C07291=1020.552,377.492,349.340,172.232,49.902,160.000
C07292=1020.561,377.739,349.299,172.241,49.902,160.002
C07293=1020.569,377.985,349.259,172.250,49.901,160.003
C07294=1020.578,378.232,349.218,172.260,49.900,160.005
C07295=1020.587,378.478,349.176,172.269,49.900,160.006
C07296=1020.595,378.724,349.136,172.279,49.900,160.007
C07297=1020.604,378.971,349.094,172.288,49.899,160.009
C07298=1020.613,379.218,349.053,172.297,49.899,160.010
C07299=1020.621,379.464,349.012,172.306,49.899,160.012
C07300=1020.630,379.710,348.971,172.315,49.898,160.013
C07301=1020.639,379.957,348.930,172.325,49.898,160.015
C07302=1020.648,380.203,348.889,172.334,49.898,160.016
C07303=1020.657,380.449,348.847,172.344,49.897,160.018
C07304=1020.665,380.696,348.806,172.353,49.897,160.019
C07305=1020.674,380.943,348.764,172.363,49.897,160.021
C07306=1020.683,381.190,348.723,172.372,49.896,160.022
C07307=1020.693,381.465,348.678,172.383,49.896,160.024
C07308=1020.703,381.741,348.632,172.394,49.896,160.025
C07309=1020.712,382.017,348.585,172.405,49.896,160.027
C07310=1020.723,382.292,348.538,172.415,49.895,160.029
C07311=1020.731,382.539,348.497,172.425,49.895,160.030
C07312=1020.740,382.786,348.455,172.435,49.895,160.032
C07313=1020.750,383.032,348.414,172.444,49.895,160.033
C07314=1020.759,383.278,348.372,172.454,49.894,160.035
C07315=1020.768,383.525,348.331,172.463,49.894,160.036
C07316=1020.777,383.771,348.289,172.473,49.894,160.038
C07317=1020.786,384.017,348.247,172.483,49.894,160.040
C07318=1020.795,384.263,348.206,172.492,49.893,160.041
C07319=1020.804,384.510,348.164,172.503,49.893,160.043
C07320=1020.813,384.756,348.123,172.513,49.893,160.044
C07321=1020.822,385.002,348.081,172.522,49.893,160.046
C07322=1020.831,385.249,348.039,172.532,49.893,160.047
C07323=1020.840,385.495,347.997,172.542,49.893,160.049
C07324=1020.849,385.741,347.955,172.551,49.893,160.051
C07325=1020.859,385.988,347.913,172.562,49.893,160.052
C07326=1020.868,386.234,347.871,172.572,49.893,160.054
C07327=1020.877,386.480,347.829,172.582,49.893,160.056
C07328=1020.886,386.726,347.786,172.592,49.893,160.057
C07329=1020.895,386.972,347.745,172.601,49.893,160.059
C07330=1020.904,387.218,347.702,172.612,49.893,160.060
C07331=1020.914,387.465,347.660,172.622,49.893,160.062
C07332=1020.923,387.711,347.618,172.632,49.893,160.064
C07333=1020.932,387.957,347.576,172.642,49.893,160.066
C07334=1020.941,388.203,347.534,172.652,49.893,160.067
C07335=1020.951,388.449,347.491,172.662,49.894,160.069
C07336=1020.959,388.696,347.449,172.672,49.894,160.071
C07337=1020.969,388.942,347.406,172.682,49.894,160.072
C07338=1020.978,389.188,347.363,172.693,49.894,160.074
C07339=1020.988,389.434,347.321,172.703,49.894,160.076
C07340=1020.996,389.680,347.278,172.713,49.894,160.078
C07341=1021.006,389.926,347.235,172.724,49.894,160.079
C07342=1021.015,390.172,347.193,172.734,49.895,160.081
C07343=1021.025,390.419,347.150,172.744,49.895,160.083
C07344=1021.034,390.664,347.107,172.754,49.895,160.084
C07345=1021.043,390.911,347.064,172.765,49.896,160.086
C07346=1021.053,391.157,347.022,172.776,49.895,160.088
C07347=1021.063,391.403,346.979,172.785,49.896,160.090
C07348=1021.072,391.648,346.936,172.796,49.897,160.092
C07349=1021.081,391.895,346.892,172.807,49.896,160.094
C07350=1021.090,392.141,346.850,172.816,49.897,160.095
C07351=1021.100,392.387,346.807,172.828,49.897,160.097
C07352=1021.110,392.632,346.764,172.838,49.897,160.099
C07353=1021.119,392.879,346.720,172.849,49.898,160.101
C07354=1021.129,393.126,346.678,172.859,49.898,160.103
C07355=1021.138,393.371,346.634,172.870,49.899,160.105
C07356=1021.147,393.618,346.591,172.880,49.899,160.106
C07357=1021.158,393.863,346.548,172.891,49.899,160.108
C07358=1021.166,394.109,346.504,172.902,49.900,160.110
C07359=1021.176,394.355,346.461,172.913,49.901,160.112
C07360=1021.186,394.601,346.417,172.923,49.901,160.114
C07361=1021.195,394.846,346.374,172.934,49.901,160.116
C07362=1021.205,395.093,346.331,172.945,49.902,160.118
C07363=1021.214,395.339,346.287,172.955,49.903,160.120
C07364=1021.225,395.585,346.243,172.967,49.903,160.122
C07365=1021.234,395.831,346.199,172.977,49.904,160.124
C07366=1021.244,396.076,346.156,172.988,49.904,160.125
C07367=1021.256,396.390,346.100,173.002,49.905,160.128
C07368=1021.268,396.703,346.045,173.016,49.906,160.131
C07369=1021.281,397.017,345.989,173.030,49.906,160.133
C07370=1021.294,397.330,345.934,173.044,49.907,160.135
C07371=1021.303,397.576,345.890,173.055,49.907,160.137
C07372=1021.313,397.822,345.845,173.067,49.908,160.140
C07373=1021.323,398.067,345.801,173.078,49.909,160.142
C07374=1021.333,398.313,345.757,173.088,49.910,160.143
C07375=1021.343,398.559,345.714,173.099,49.910,160.145
C07376=1021.352,398.805,345.669,173.111,49.911,160.148
C07377=1021.363,399.051,345.625,173.122,49.912,160.150
C07378=1021.372,399.297,345.581,173.134,49.913,160.152
C07379=1021.382,399.542,345.536,173.144,49.913,160.154
C07380=1021.392,399.788,345.493,173.155,49.914,160.156
C07381=1021.402,400.034,345.448,173.167,49.915,160.158
C07382=1021.412,400.280,345.403,173.179,49.916,160.160
C07383=1021.422,400.526,345.359,173.190,49.916,160.162
C07384=1021.432,400.771,345.314,173.202,49.917,160.164
C07385=1021.441,401.017,345.270,173.213,49.918,160.166
C07386=1021.452,401.263,345.226,173.225,49.919,160.169
C07387=1021.462,401.509,345.181,173.236,49.920,160.171
C07388=1021.472,401.754,345.136,173.248,49.921,160.173
C07389=1021.481,402.000,345.091,173.259,49.922,160.175
C07390=1021.492,402.246,345.046,173.271,49.922,160.177
C07391=1021.501,402.491,345.001,173.282,49.923,160.179
C07392=1021.512,402.737,344.957,173.294,49.924,160.181
C07393=1021.522,402.983,344.912,173.306,49.925,160.184
C07394=1021.532,403.228,344.867,173.317,49.926,160.186
C07395=1021.542,403.475,344.822,173.329,49.927,160.188
C07396=1021.552,403.720,344.777,173.341,49.928,160.190
C07397=1021.563,403.965,344.732,173.352,49.929,160.192
C07398=1021.573,404.211,344.687,173.364,49.931,160.195
C07399=1021.583,404.456,344.642,173.376,49.932,160.197
C07400=1021.593,404.702,344.596,173.388,49.933,160.199
C07401=1021.604,404.948,344.551,173.399,49.934,160.202
C07402=1021.613,405.194,344.506,173.412,49.935,160.204
C07403=1021.625,405.439,344.461,173.424,49.936,160.206
C07404=1021.634,405.684,344.416,173.436,49.937,160.208
C07405=1021.645,405.930,344.370,173.448,49.939,160.211
C07406=1021.655,406.176,344.325,173.460,49.939,160.213
C07407=1021.666,406.422,344.279,173.472,49.941,160.216
C07408=1021.677,406.666,344.234,173.484,49.942,160.218
C07409=1021.687,406.913,344.189,173.496,49.943,160.220
C07410=1021.698,407.158,344.143,173.509,49.944,160.222
C07411=1021.708,407.404,344.097,173.521,49.945,160.225
C07412=1021.719,407.650,344.052,173.533,49.946,160.227
C07413=1021.729,407.895,344.006,173.545,49.948,160.230
C07414=1021.740,408.140,343.961,173.557,49.949,160.232
C07415=1021.751,408.386,343.915,173.570,49.950,160.234
C07416=1021.761,408.631,343.869,173.582,49.951,160.237
C07417=1021.772,408.877,343.823,173.595,49.952,160.239
C07418=1021.782,409.123,343.777,173.607,49.954,160.242
C07419=1021.793,409.368,343.731,173.620,49.955,160.244
C07420=1021.804,409.614,343.686,173.632,49.957,160.246
C07421=1021.815,409.859,343.639,173.645,49.958,160.249
C07422=1021.825,410.104,343.593,173.657,49.959,160.251
C07423=1021.836,410.350,343.547,173.671,49.961,160.254
C07424=1021.846,410.595,343.500,173.683,49.963,160.256
C07425=1021.857,410.841,343.454,173.696,49.964,160.259
C07426=1021.868,411.086,343.407,173.708,49.965,160.261
C07427=1021.881,411.399,343.348,173.724,49.968,160.265
C07428=1021.895,411.712,343.289,173.741,49.969,160.268
C07429=1021.910,412.026,343.230,173.757,49.971,160.271
C07430=1021.923,412.338,343.171,173.773,49.973,160.274
C07431=1021.934,412.584,343.124,173.786,49.975,160.277
C07432=1021.945,412.829,343.077,173.799,49.976,160.280
C07433=1021.956,413.074,343.031,173.813,49.978,160.282
C07434=1021.967,413.320,342.984,173.825,49.979,160.285
C07435=1021.978,413.565,342.937,173.838,49.981,160.287
C07436=1021.989,413.810,342.890,173.852,49.983,160.290
C07437=1022.000,414.055,342.843,173.865,49.984,160.293
C07438=1022.011,414.300,342.797,173.878,49.986,160.295
C07439=1022.022,414.546,342.749,173.892,49.987,160.298
C07440=1022.033,414.791,342.702,173.904,49.989,160.301
C07441=1022.045,415.037,342.655,173.917,49.991,160.303
C07442=1022.056,415.283,342.608,173.931,49.993,160.306
C07443=1022.067,415.528,342.562,173.944,49.994,160.309
C07444=1022.078,415.773,342.514,173.958,49.996,160.312
C07445=1022.089,416.018,342.467,173.971,49.998,160.314
C07446=1022.100,416.263,342.419,173.985,49.999,160.317
C07447=1022.112,416.509,342.372,173.998,50.002,160.320
C07448=1022.122,416.754,342.324,174.012,50.003,160.323
C07449=1022.134,416.999,342.277,174.025,50.005,160.325
C07450=1022.146,417.244,342.229,174.039,50.007,160.328
C07451=1022.156,417.489,342.181,174.052,50.009,160.331
C07452=1022.168,417.735,342.134,174.067,50.011,160.334
C07453=1022.179,417.980,342.086,174.081,50.013,160.337
C07454=1022.191,418.225,342.038,174.094,50.015,160.340
C07455=1022.202,418.470,341.990,174.108,50.016,160.342
C07456=1022.213,418.716,341.942,174.122,50.019,160.345
C07457=1022.225,418.960,341.895,174.136,50.021,160.348
C07458=1022.236,419.205,341.846,174.150,50.022,160.351
C07459=1022.248,419.450,341.799,174.164,50.024,160.354
C07460=1022.259,419.695,341.751,174.177,50.027,160.357
C07461=1022.271,419.941,341.703,174.192,50.028,160.360
C07462=1022.282,420.186,341.655,174.206,50.031,160.363
C07463=1022.294,420.432,341.606,174.221,50.033,160.366
C07464=1022.306,420.676,341.558,174.235,50.035,160.369
C07465=1022.318,420.921,341.510,174.249,50.037,160.372
C07466=1022.329,421.167,341.462,174.263,50.039,160.375
C07467=1022.341,421.411,341.414,174.277,50.041,160.378
C07468=1022.352,421.657,341.365,174.292,50.043,160.381
C07469=1022.365,421.902,341.316,174.306,50.045,160.384
C07470=1022.376,422.147,341.268,174.321,50.047,160.387
C07471=1022.389,422.415,341.215,174.336,50.050,160.390
C07472=1022.402,422.683,341.161,174.352,50.052,160.393
C07473=1022.415,422.951,341.108,174.369,50.054,160.397
C07474=1022.428,423.219,341.055,174.384,50.057,160.400
C07475=1022.439,423.463,341.006,174.399,50.059,160.403
C07476=1022.451,423.709,340.957,174.414,50.062,160.407
C07477=1022.464,423.953,340.908,174.428,50.064,160.410
C07478=1022.476,424.199,340.859,174.443,50.066,160.413
C07479=1022.488,424.443,340.810,174.459,50.068,160.416
C07480=1022.500,424.689,340.761,174.474,50.071,160.419
C07481=1022.511,424.933,340.712,174.488,50.073,160.422
C07482=1022.524,425.178,340.662,174.503,50.076,160.426
C07483=1022.536,425.423,340.613,174.518,50.078,160.429
C07484=1022.548,425.668,340.564,174.534,50.080,160.432
C07485=1022.560,425.913,340.514,174.549,50.083,160.435
C07486=1022.572,426.157,340.466,174.564,50.085,160.439
C07487=1022.588,426.479,340.400,174.584,50.089,160.443
C07488=1022.604,426.800,340.335,174.604,50.091,160.447
C07489=1022.620,427.120,340.269,174.624,50.095,160.452
C07490=1022.636,427.441,340.204,174.644,50.098,160.456
C07491=1022.648,427.685,340.155,174.660,50.101,160.459
C07492=1022.661,427.930,340.105,174.675,50.103,160.463
C07493=1022.673,428.175,340.055,174.691,50.106,160.466
C07494=1022.685,428.420,340.004,174.706,50.109,160.470
C07495=1022.697,428.665,339.954,174.722,50.111,160.473
C07496=1022.710,428.909,339.904,174.738,50.114,160.476
C07497=1022.723,429.154,339.855,174.754,50.116,160.480
C07498=1022.735,429.399,339.805,174.769,50.119,160.483
C07499=1022.747,429.643,339.755,174.785,50.122,160.487
C07500=1022.760,429.888,339.704,174.802,50.125,160.490
C07501=1022.772,430.133,339.654,174.817,50.127,160.494
C07502=1022.785,430.377,339.604,174.834,50.130,160.497
C07503=1022.799,430.622,339.553,174.849,50.133,160.501
C07504=1022.811,430.867,339.503,174.866,50.135,160.504
C07505=1022.824,431.111,339.452,174.881,50.138,160.508
C07506=1022.836,431.355,339.401,174.898,50.141,160.511
C07507=1022.849,431.601,339.351,174.914,50.144,160.515
C07508=1022.862,431.845,339.300,174.931,50.147,160.519
C07509=1022.875,432.089,339.250,174.947,50.149,160.522
C07510=1022.888,432.334,339.199,174.964,50.152,160.526
C07511=1022.901,432.578,339.149,174.980,50.155,160.529
C07512=1022.914,432.823,339.097,174.997,50.158,160.533
C07513=1022.927,433.067,339.046,175.013,50.161,160.537
C07514=1022.939,433.311,338.995,175.030,50.164,160.540
C07515=1022.953,433.556,338.944,175.047,50.166,160.544
C07516=1022.965,433.800,338.893,175.064,50.169,160.548
C07517=1022.978,434.045,338.842,175.081,50.172,160.552
C07518=1022.992,434.289,338.790,175.097,50.176,160.555
C07519=1023.005,434.534,338.739,175.114,50.179,160.559
C07520=1023.018,434.778,338.687,175.131,50.182,160.563
C07521=1023.031,435.023,338.635,175.148,50.185,160.567
C07522=1023.044,435.267,338.584,175.165,50.188,160.571
C07523=1023.057,435.512,338.533,175.182,50.191,160.574
C07524=1023.070,435.756,338.481,175.199,50.194,160.578
C07525=1023.084,436.000,338.429,175.217,50.197,160.582
C07526=1023.097,436.244,338.377,175.235,50.200,160.586
C07527=1023.110,436.488,338.326,175.252,50.203,160.590
C07528=1023.124,436.732,338.274,175.269,50.207,160.594
C07529=1023.137,436.977,338.222,175.286,50.210,160.598
C07530=1023.150,437.221,338.169,175.304,50.212,160.602
C07531=1023.164,437.465,338.117,175.322,50.216,160.606
C07532=1023.177,437.710,338.066,175.339,50.219,160.610
C07533=1023.191,437.954,338.014,175.357,50.222,160.614
C07534=1023.204,438.198,337.961,175.375,50.226,160.618
C07535=1022.814,436.266,338.039,175.226,50.266,160.605
C07536=1022.801,436.022,338.091,175.209,50.264,160.601
C07537=1022.788,435.777,338.142,175.191,50.260,160.597
C07538=1022.774,435.533,338.194,175.174,50.257,160.593
C07539=1022.761,435.289,338.246,175.157,50.254,160.589
C07540=1022.748,435.044,338.297,175.139,50.252,160.585
C07541=1022.735,434.800,338.349,175.122,50.248,160.581
C07542=1022.722,434.556,338.400,175.105,50.245,160.578
C07543=1022.708,434.312,338.451,175.088,50.243,160.574
C07544=1022.695,434.067,338.503,175.071,50.240,160.570
C07545=1022.683,433.823,338.553,175.054,50.237,160.567
C07546=1022.669,433.578,338.605,175.038,50.234,160.563
C07547=1022.656,433.334,338.656,175.021,50.231,160.559
C07548=1022.643,433.089,338.707,175.004,50.228,160.555
C07549=1022.631,432.845,338.758,174.988,50.226,160.552
C07550=1022.618,432.601,338.809,174.971,50.223,160.548
C07551=1022.605,432.356,338.860,174.955,50.220,160.544
C07552=1022.592,432.112,338.911,174.938,50.217,160.541
C07553=1022.579,431.867,338.962,174.922,50.215,160.537
C07554=1022.567,431.622,339.012,174.905,50.212,160.534
C07555=1022.554,431.378,339.063,174.889,50.209,160.530
C07556=1022.540,431.133,339.114,174.873,50.206,160.526
C07557=1022.528,430.888,339.164,174.857,50.204,160.523
C07558=1022.515,430.644,339.214,174.840,50.201,160.519
C07559=1022.503,430.399,339.265,174.825,50.198,160.516
C07560=1022.490,430.154,339.315,174.808,50.196,160.512
C07561=1022.477,429.911,339.365,174.792,50.193,160.509
C07562=1022.464,429.665,339.415,174.776,50.191,160.505
C07563=1022.452,429.420,339.465,174.760,50.188,160.502
C07564=1022.439,429.176,339.516,174.744,50.186,160.499
C07565=1022.427,428.931,339.566,174.729,50.183,160.495
C07566=1022.415,428.686,339.616,174.713,50.180,160.492
C07567=1022.402,428.442,339.666,174.697,50.178,160.488
C07568=1022.390,428.198,339.716,174.681,50.176,160.485
C07569=1022.378,427.953,339.766,174.666,50.173,160.482
C07570=1022.365,427.708,339.816,174.650,50.170,160.478
C07571=1022.353,427.463,339.865,174.635,50.168,160.475
C07572=1022.338,427.163,339.926,174.616,50.165,160.471
C07573=1022.323,426.862,339.988,174.596,50.162,160.467
C07574=1022.308,426.561,340.048,174.578,50.159,160.463
C07575=1022.294,426.261,340.110,174.559,50.156,160.458
C07576=1022.281,426.016,340.159,174.543,50.154,160.455
C07577=1022.269,425.771,340.208,174.528,50.152,160.452
C07578=1022.257,425.526,340.258,174.513,50.149,160.449
C07579=1022.245,425.281,340.308,174.498,50.147,160.445
C07580=1022.233,425.037,340.356,174.483,50.145,160.442
C07581=1022.221,424.791,340.406,174.468,50.143,160.439
C07582=1022.209,424.546,340.455,174.454,50.140,160.436
C07583=1022.197,424.301,340.503,174.438,50.138,160.433
C07584=1022.185,424.057,340.552,174.424,50.136,160.430
C07585=1022.172,423.811,340.601,174.408,50.134,160.426
C07586=1022.161,423.567,340.650,174.394,50.132,160.423
C07587=1022.149,423.321,340.700,174.379,50.129,160.420
C07588=1022.137,423.077,340.748,174.364,50.127,160.417
C07589=1022.125,422.832,340.797,174.349,50.125,160.414
C07590=1022.113,422.587,340.846,174.335,50.123,160.411
C07591=1022.102,422.342,340.894,174.321,50.121,160.408
C07592=1022.090,422.097,340.943,174.305,50.119,160.405
C07593=1022.078,421.852,340.992,174.292,50.116,160.402
C07594=1022.067,421.607,341.040,174.277,50.115,160.399
C07595=1022.055,421.362,341.089,174.263,50.112,160.396
C07596=1022.043,421.116,341.137,174.248,50.111,160.393
C07597=1022.031,420.872,341.185,174.234,50.108,160.390
C07598=1022.020,420.627,341.234,174.220,50.107,160.387
C07599=1022.008,420.382,341.281,174.206,50.104,160.384
C07600=1021.996,420.137,341.329,174.191,50.103,160.381
C07601=1021.985,419.891,341.377,174.177,50.100,160.378
C07602=1021.973,419.647,341.426,174.163,50.099,160.375
C07603=1021.962,419.401,341.474,174.149,50.097,160.372
C07604=1021.950,419.156,341.522,174.135,50.095,160.369
C07605=1021.938,418.911,341.570,174.121,50.093,160.366
C07606=1021.927,418.666,341.618,174.107,50.091,160.364
C07607=1021.916,418.420,341.665,174.093,50.090,160.361
C07608=1021.904,418.175,341.713,174.078,50.088,160.358
C07609=1021.893,417.930,341.761,174.065,50.086,160.355
C07610=1021.881,417.685,341.808,174.051,50.084,160.352
C07611=1021.870,417.440,341.856,174.038,50.082,160.349
C07612=1021.859,417.194,341.903,174.024,50.081,160.347
C07613=1021.848,416.949,341.952,174.010,50.079,160.344
C07614=1021.837,416.704,341.998,173.996,50.077,160.341
C07615=1021.825,416.459,342.046,173.983,50.075,160.338
C07616=1021.814,416.213,342.094,173.969,50.074,160.335
C07617=1021.803,415.969,342.141,173.956,50.072,160.333
C07618=1021.792,415.723,342.189,173.942,50.070,160.330
C07619=1021.780,415.478,342.236,173.929,50.069,160.327
C07620=1021.764,415.118,342.305,173.909,50.066,160.323
C07621=1021.748,414.757,342.375,173.890,50.064,160.319
C07622=1021.731,414.397,342.443,173.870,50.062,160.315
C07623=1021.715,414.036,342.512,173.851,50.059,160.311
C07624=1021.704,413.791,342.559,173.838,50.057,160.309
C07625=1021.693,413.546,342.606,173.825,50.056,160.306
C07626=1021.682,413.301,342.652,173.811,50.054,160.304
C07627=1021.671,413.056,342.699,173.798,50.053,160.301
C07628=1021.660,412.821,342.744,173.786,50.051,160.298
C07629=1021.650,412.587,342.788,173.773,50.050,160.296
C07630=1021.639,412.352,342.833,173.761,50.049,160.293
C07631=1021.629,412.118,342.878,173.749,50.047,160.291
C07632=1021.619,411.884,342.922,173.736,50.046,160.289
C07633=1021.608,411.648,342.966,173.724,50.045,160.286
C07634=1021.598,411.414,343.010,173.712,50.044,160.284
C07635=1021.588,411.180,343.055,173.700,50.042,160.281
C07636=1021.578,410.935,343.101,173.687,50.041,160.279
C07637=1021.567,410.690,343.147,173.673,50.039,160.276
C07638=1021.555,410.443,343.194,173.661,50.038,160.274
C07639=1021.545,410.198,343.240,173.648,50.037,160.271
C07640=1021.534,409.953,343.286,173.636,50.035,160.269
C07641=1021.524,409.707,343.333,173.623,50.034,160.266
C07642=1021.513,409.461,343.379,173.610,50.033,160.264
C07643=1021.502,409.216,343.425,173.598,50.031,160.261
C07644=1021.492,408.971,343.471,173.585,50.030,160.259
C07645=1021.481,408.725,343.517,173.573,50.029,160.257
C07646=1021.471,408.479,343.562,173.560,50.028,160.254
C07647=1021.460,408.234,343.608,173.548,50.026,160.252
C07648=1021.449,407.988,343.653,173.536,50.026,160.250
C07649=1021.438,407.742,343.699,173.524,50.024,160.247
C07650=1021.428,407.497,343.745,173.511,50.023,160.245
C07651=1021.418,407.252,343.791,173.499,50.022,160.242
C07652=1021.407,407.006,343.836,173.487,50.021,160.240
C07653=1021.396,406.760,343.881,173.474,50.020,160.238
C07654=1021.385,406.515,343.927,173.463,50.019,160.235
C07655=1021.376,406.269,343.972,173.451,50.018,160.233
C07656=1021.365,406.024,344.018,173.438,50.017,160.231
C07657=1021.355,405.777,344.063,173.426,50.016,160.229
C07658=1021.344,405.533,344.108,173.414,50.014,160.226
C07659=1021.334,405.287,344.153,173.402,50.014,160.224
C07660=1021.323,405.041,344.199,173.390,50.013,160.222
C07661=1021.313,404.796,344.244,173.378,50.012,160.219
C07662=1021.303,404.549,344.289,173.367,50.011,160.217
C07663=1021.292,404.305,344.334,173.353,50.010,160.215
C07664=1021.282,404.059,344.379,173.342,50.009,160.212
C07665=1021.272,403.813,344.424,173.330,50.008,160.210
C07666=1021.262,403.567,344.469,173.318,50.007,160.208
C07667=1021.252,403.321,344.514,173.307,50.006,160.206
C07668=1021.242,403.076,344.558,173.295,50.005,160.204
C07669=1021.231,402.830,344.604,173.284,50.004,160.202
C07670=1021.221,402.585,344.649,173.271,50.004,160.199
C07671=1021.212,402.339,344.694,173.260,50.003,160.197
C07672=1021.201,402.093,344.739,173.248,50.002,160.195
C07673=1021.192,401.847,344.783,173.236,50.001,160.193
C07674=1021.181,401.602,344.827,173.225,50.000,160.191
C07675=1021.171,401.356,344.873,173.213,49.999,160.189
C07676=1021.161,401.110,344.917,173.202,49.998,160.186
C07677=1021.152,400.865,344.962,173.190,49.998,160.184
C07678=1021.142,400.619,345.006,173.179,49.997,160.182
C07679=1021.132,400.373,345.051,173.167,49.996,160.180
C07680=1021.122,400.127,345.096,173.156,49.995,160.178
C07681=1021.111,399.881,345.139,173.145,49.995,160.176
C07682=1021.102,399.636,345.184,173.134,49.994,160.174
C07683=1021.092,399.390,345.228,173.123,49.993,160.172
C07684=1021.082,399.144,345.273,173.111,49.993,160.170
C07685=1021.072,398.898,345.317,173.100,49.992,160.168
C07686=1021.062,398.652,345.360,173.088,49.991,160.166
C07687=1021.053,398.407,345.405,173.077,49.991,160.164
C07688=1021.043,398.161,345.449,173.066,49.991,160.162
C07689=1021.033,397.915,345.493,173.055,49.990,160.160
C07690=1021.024,397.669,345.537,173.044,49.989,160.158
C07691=1021.013,397.423,345.580,173.033,49.988,160.155
C07692=1021.001,397.108,345.637,173.019,49.988,160.153
C07693=1020.988,396.792,345.694,173.004,49.987,160.150
C07694=1020.975,396.477,345.749,172.990,49.986,160.148
C07695=1020.963,396.161,345.805,172.976,49.986,160.146
C07696=1020.953,395.915,345.848,172.965,49.986,160.144
C07697=1020.944,395.669,345.892,172.954,49.985,160.142
C07698=1020.934,395.424,345.936,172.943,49.984,160.140
C07699=1020.925,395.177,345.980,172.932,49.985,160.138
C07700=1020.914,394.932,346.023,172.921,49.984,160.136
C07701=1020.905,394.685,346.066,172.911,49.983,160.134
C07702=1020.896,394.440,346.110,172.900,49.983,160.132
C07703=1020.886,394.194,346.153,172.889,49.983,160.130
C07704=1020.877,393.947,346.197,172.878,49.982,160.128
C07705=1020.867,393.702,346.240,172.868,49.982,160.126
C07706=1020.857,393.456,346.283,172.857,49.981,160.125
C07707=1020.848,393.209,346.327,172.846,49.982,160.123
C07708=1020.839,392.964,346.369,172.836,49.981,160.121
C07709=1020.829,392.718,346.413,172.825,49.981,160.119
C07710=1020.820,392.472,346.456,172.814,49.981,160.117
C07711=1020.810,392.225,346.498,172.804,49.980,160.115
C07712=1020.800,391.979,346.541,172.793,49.980,160.114
C07713=1020.791,391.734,346.585,172.783,49.980,160.112
C07714=1020.782,391.487,346.628,172.772,49.980,160.110
C07715=1020.772,391.241,346.670,172.762,49.979,160.108
C07716=1020.762,390.995,346.713,172.751,49.980,160.106
C07717=1020.754,390.749,346.756,172.741,49.979,160.105
C07718=1020.744,390.502,346.799,172.731,49.979,160.103
C07719=1020.735,390.257,346.841,172.720,49.979,160.101
C07720=1020.726,390.011,346.884,172.711,49.979,160.100
C07721=1020.716,389.764,346.926,172.699,49.978,160.098
C07722=1020.707,389.518,346.970,172.689,49.978,160.096
C07723=1020.697,389.272,347.012,172.679,49.978,160.094
C07724=1020.688,389.026,347.055,172.669,49.979,160.093
C07725=1020.679,388.780,347.097,172.659,49.978,160.091
C07726=1020.671,388.534,347.139,172.648,49.979,160.089
C07727=1020.661,388.287,347.182,172.638,49.978,160.087
C07728=1020.652,388.042,347.225,172.628,49.978,160.086
C07729=1020.643,387.795,347.266,172.617,49.978,160.084
C07730=1020.633,387.549,347.309,172.608,49.979,160.082
C07731=1020.624,387.303,347.352,172.598,49.978,160.081
C07732=1020.615,387.057,347.393,172.588,49.978,160.079
C07733=1020.606,386.811,347.436,172.578,49.979,160.077
C07734=1020.597,386.565,347.478,172.568,49.979,160.076
C07735=1020.588,386.318,347.519,172.558,49.978,160.074
C07736=1020.578,386.072,347.562,172.547,49.979,160.073
C07737=1020.569,385.825,347.604,172.537,49.979,160.071
C07738=1020.560,385.580,347.646,172.528,49.979,160.069
C07739=1020.551,385.333,347.688,172.518,49.979,160.068
C07740=1020.542,385.087,347.730,172.508,49.979,160.066
C07741=1020.533,384.841,347.771,172.498,49.980,160.065
C07742=1020.524,384.594,347.813,172.488,49.980,160.063
C07743=1020.515,384.348,347.855,172.479,49.980,160.061
C07744=1020.505,384.102,347.896,172.469,49.980,160.060
C07745=1020.496,383.855,347.938,172.459,49.980,160.058
C07746=1020.487,383.609,347.979,172.449,49.981,160.057
C07747=1020.478,383.363,348.021,172.439,49.981,160.055
C07748=1020.470,383.116,348.063,172.430,49.981,160.054
C07749=1020.461,382.870,348.104,172.420,49.982,160.052
C07750=1020.451,382.624,348.146,172.411,49.982,160.051
C07751=1020.442,382.378,348.187,172.401,49.982,160.049
C07752=1020.432,382.100,348.234,172.390,49.983,160.047
C07753=1020.423,381.821,348.280,172.379,49.983,160.046
C07754=1020.412,381.542,348.327,172.368,49.984,160.044
C07755=1020.402,381.264,348.374,172.357,49.984,160.042
C07756=1020.393,381.018,348.416,172.347,49.984,160.041
C07757=1020.385,380.771,348.456,172.338,49.984,160.039
C07758=1020.375,380.525,348.497,172.329,49.985,160.038
C07759=1020.366,380.279,348.539,172.319,49.986,160.036
C07760=1020.358,380.032,348.580,172.310,49.986,160.035
C07761=1020.349,379.786,348.621,172.300,49.986,160.033
C07762=1020.341,379.539,348.662,172.291,49.987,160.032
C07763=1020.331,379.293,348.703,172.281,49.988,160.031
C07764=1020.323,379.047,348.744,172.272,49.988,160.029
C07765=1020.315,378.800,348.785,172.262,49.988,160.028
C07766=1020.306,378.554,348.827,172.253,49.989,160.026
C07767=1020.298,378.307,348.868,172.245,49.989,160.025
C07768=1020.289,378.060,348.909,172.235,49.989,160.023
C07769=1020.280,377.814,348.949,172.226,49.990,160.022
C07770=1020.271,377.568,348.990,172.216,49.991,160.021
C07771=1020.263,377.322,349.031,172.207,49.991,160.019
C07772=1020.255,377.075,349.072,172.198,49.992,160.018
C07773=1020.247,376.828,349.113,172.188,49.992,160.016
C07774=1020.237,376.582,349.153,172.179,49.993,160.015
C07775=1020.229,376.335,349.194,172.171,49.994,160.014
C07776=1020.220,376.089,349.235,172.161,49.994,160.012
C07777=1020.212,375.842,349.275,172.152,49.995,160.011
C07778=1020.203,375.595,349.316,172.143,49.995,160.010
C07779=1020.194,375.350,349.356,172.134,49.996,160.008
C07780=1020.186,375.103,349.397,172.125,49.997,160.007
C07781=1020.177,374.857,349.437,172.115,49.998,160.006
C07782=1020.169,374.609,349.477,172.107,49.999,160.005
C07783=1020.160,374.363,349.517,172.098,49.999,160.003
C07784=1020.152,374.117,349.558,172.089,50.000,160.002
C07785=1020.143,373.869,349.597,172.079,50.001,160.001
C07786=1020.135,373.623,349.638,172.070,50.002,159.999
C07787=1020.126,373.377,349.678,172.062,50.002,159.998
C07788=1020.118,373.130,349.718,172.053,50.003,159.997
C07789=1020.109,372.884,349.758,172.044,50.004,159.996
C07790=1020.101,372.637,349.798,172.035,50.005,159.994
C07791=1020.092,372.390,349.839,172.027,50.006,159.993
C07792=1020.083,372.143,349.878,172.017,50.007,159.992
C07793=1020.075,371.897,349.919,172.008,50.007,159.990
C07794=1020.067,371.651,349.958,172.000,50.008,159.989
C07795=1020.059,371.404,349.998,171.991,50.009,159.988
C07796=1020.050,371.157,350.038,171.982,50.010,159.987
C07797=1020.042,370.910,350.078,171.973,50.011,159.986
C07798=1020.034,370.663,350.118,171.965,50.012,159.984
C07799=1020.026,370.417,350.158,171.956,50.013,159.983
C07800=1020.017,370.171,350.198,171.947,50.014,159.982
C07801=1020.009,369.924,350.237,171.939,50.015,159.981
C07802=1020.001,369.677,350.277,171.930,50.016,159.980
C07803=1019.993,369.430,350.317,171.922,50.016,159.978
C07804=1019.985,369.184,350.356,171.913,50.018,159.977
C07805=1019.976,368.938,350.396,171.904,50.019,159.976
C07806=1019.968,368.691,350.436,171.896,50.019,159.975
C07807=1019.960,368.444,350.475,171.887,50.021,159.974
C07808=1019.952,368.197,350.515,171.879,50.021,159.973
C07809=1019.944,367.951,350.555,171.870,50.023,159.971
C07810=1019.936,367.704,350.594,171.861,50.024,159.970
C07811=1019.928,367.456,350.633,171.853,50.025,159.969
C07812=1019.918,367.200,350.674,171.844,50.026,159.968
C07813=1019.910,366.945,350.715,171.835,50.028,159.967
C07814=1019.902,366.689,350.756,171.826,50.029,159.966
C07815=1019.894,366.433,350.796,171.817,50.030,159.964
C07816=1019.885,366.186,350.835,171.809,50.031,159.963
C07817=1019.877,365.939,350.874,171.801,50.033,159.962
C07818=1019.869,365.692,350.913,171.792,50.033,159.961
C07819=1019.860,365.445,350.952,171.784,50.035,159.960
C07820=1019.852,365.199,350.992,171.776,50.036,159.959
C07821=1019.844,364.951,351.030,171.767,50.037,159.958
C07822=1019.835,364.705,351.069,171.759,50.039,159.957
C07823=1019.828,364.458,351.108,171.750,50.039,159.956
C07824=1019.820,364.211,351.148,171.742,50.041,159.955
C07825=1019.812,363.964,351.186,171.734,50.042,159.954
C07826=1019.804,363.717,351.225,171.726,50.043,159.953
C07827=1019.796,363.471,351.264,171.717,50.045,159.952
C07828=1019.788,363.224,351.302,171.709,50.046,159.951
C07829=1019.780,362.977,351.341,171.701,50.048,159.950
C07830=1019.772,362.731,351.380,171.693,50.049,159.949
C07831=1019.764,362.483,351.419,171.684,50.050,159.947
C07832=1019.756,362.236,351.458,171.676,50.051,159.946
C07833=1019.749,361.989,351.496,171.667,50.053,159.945
C07834=1019.740,361.743,351.535,171.660,50.054,159.944
C07835=1019.732,361.496,351.574,171.652,50.056,159.944
C07836=1019.724,361.249,351.612,171.644,50.057,159.943
C07837=1019.716,361.002,351.651,171.636,50.059,159.942
C07838=1019.709,360.755,351.689,171.627,50.060,159.940
C07839=1019.701,360.508,351.728,171.619,50.061,159.939
C07840=1019.693,360.261,351.767,171.611,50.062,159.938
C07841=1019.686,360.014,351.805,171.603,50.064,159.938
C07842=1019.677,359.767,351.844,171.595,50.066,159.937
C07843=1019.670,359.520,351.882,171.588,50.067,159.936
C07844=1019.662,359.273,351.921,171.579,50.069,159.935
C07845=1019.654,359.027,351.959,171.571,50.070,159.934
C07846=1019.646,358.779,351.997,171.564,50.072,159.933
C07847=1019.638,358.533,352.034,171.555,50.073,159.932
C07848=1019.631,358.286,352.073,171.547,50.075,159.931
C07849=1019.622,358.039,352.111,171.539,50.077,159.930
C07850=1019.615,357.792,352.149,171.531,50.078,159.929
C07851=1019.607,357.545,352.187,171.524,50.080,159.928
C07852=1019.599,357.298,352.226,171.515,50.082,159.927
C07853=1019.591,357.050,352.263,171.508,50.083,159.926
C07854=1019.583,356.804,352.301,171.500,50.085,159.926
C07855=1019.576,356.557,352.339,171.492,50.086,159.924
C07856=1019.568,356.310,352.377,171.484,50.088,159.924
C07857=1019.560,356.063,352.415,171.477,50.090,159.923
C07858=1019.552,355.816,352.452,171.469,50.091,159.922
C07859=1019.545,355.568,352.490,171.461,50.093,159.921
C07860=1019.537,355.322,352.529,171.453,50.095,159.920
C07861=1019.530,355.075,352.566,171.446,50.097,159.919
C07862=1019.522,354.828,352.605,171.437,50.098,159.918
C07863=1019.514,354.581,352.642,171.430,50.100,159.917
C07864=1019.506,354.334,352.679,171.422,50.102,159.917
C07865=1019.499,354.087,352.717,171.415,50.104,159.916
C07866=1019.492,353.840,352.755,171.406,50.106,159.915
C07867=1019.483,353.592,352.792,171.399,50.107,159.914
C07868=1019.476,353.345,352.830,171.392,50.109,159.913
C07869=1019.468,353.098,352.867,171.384,50.111,159.913
C07870=1019.460,352.851,352.904,171.376,50.113,159.912
C07871=1019.453,352.605,352.942,171.368,50.115,159.911
C07872=1019.445,352.356,352.980,171.361,50.117,159.910
C07873=1019.437,352.107,353.017,171.354,50.118,159.909
C07874=1019.429,351.858,353.055,171.345,50.121,159.909
C07875=1019.422,351.609,353.092,171.338,50.122,159.908
C07876=1019.414,351.362,353.129,171.330,50.124,159.907
C07877=1019.407,351.115,353.167,171.323,50.126,159.906
C07878=1019.399,350.868,353.204,171.315,50.128,159.905
C07879=1019.392,350.621,353.241,171.307,50.130,159.904
C07880=1019.384,350.374,353.278,171.300,50.132,159.904
C07881=1019.377,350.127,353.316,171.293,50.134,159.903
C07882=1019.369,349.880,353.353,171.286,50.136,159.902
C07883=1019.362,349.633,353.390,171.278,50.138,159.901
C07884=1019.354,349.386,353.427,171.270,50.140,159.901
C07885=1019.347,349.139,353.464,171.263,50.142,159.900
C07886=1019.339,348.892,353.502,171.255,50.144,159.899
C07887=1019.332,348.644,353.538,171.248,50.146,159.898
C07888=1019.324,348.397,353.575,171.241,50.148,159.898
C07889=1019.317,348.150,353.613,171.233,50.150,159.897
C07890=1019.309,347.902,353.649,171.226,50.152,159.896
C07891=1019.302,347.655,353.687,171.218,50.154,159.896
C07892=1019.295,347.408,353.723,171.211,50.156,159.895
C07893=1019.287,347.161,353.760,171.204,50.159,159.894
C07894=1019.280,346.915,353.797,171.196,50.160,159.893
C07895=1019.273,346.667,353.834,171.189,50.163,159.893
C07896=1019.265,346.419,353.870,171.182,50.165,159.892
C07897=1019.257,346.173,353.907,171.175,50.167,159.891
C07898=1019.250,345.925,353.944,171.168,50.169,159.891
C07899=1019.243,345.677,353.980,171.159,50.171,159.890
C07900=1019.235,345.431,354.016,171.152,50.174,159.889
C07901=1019.228,345.184,354.053,171.145,50.176,159.889
C07902=1019.221,344.936,354.089,171.138,50.178,159.888
C07903=1019.213,344.689,354.126,171.131,50.181,159.887
C07904=1019.206,344.442,354.163,171.124,50.183,159.887
C07905=1019.199,344.195,354.199,171.117,50.185,159.886
C07906=1019.191,343.947,354.235,171.110,50.187,159.885
C07907=1019.184,343.700,354.272,171.103,50.190,159.885
C07908=1019.177,343.453,354.308,171.096,50.192,159.884
C07909=1019.169,343.206,354.345,171.088,50.194,159.883
C07910=1019.161,342.959,354.381,171.081,50.196,159.883
C07911=1019.155,342.712,354.418,171.073,50.199,159.882
C07912=1019.147,342.464,354.454,171.066,50.201,159.882
C07913=1019.140,342.217,354.490,171.059,50.204,159.881
C07914=1019.133,341.970,354.526,171.052,50.206,159.880
C07915=1019.126,341.722,354.563,171.045,50.209,159.880
C07916=1019.118,341.475,354.599,171.038,50.211,159.879
C07917=1019.111,341.227,354.634,171.031,50.213,159.879
C07918=1019.104,340.980,354.670,171.024,50.216,159.878
C07919=1019.097,340.733,354.707,171.017,50.218,159.877
C07920=1019.090,340.485,354.743,171.010,50.221,159.877
C07921=1019.082,340.239,354.779,171.003,50.223,159.876
C07922=1019.075,339.991,354.815,170.996,50.225,159.876
C07923=1019.069,339.743,354.851,170.989,50.228,159.875
C07924=1019.061,339.496,354.887,170.982,50.230,159.874
C07925=1019.054,339.249,354.923,170.975,50.233,159.874
C07926=1019.046,339.002,354.959,170.968,50.235,159.873
C07927=1019.040,338.754,354.994,170.961,50.237,159.873
C07928=1019.032,338.507,355.030,170.954,50.240,159.872
C07929=1019.025,338.260,355.065,170.947,50.243,159.872
C07930=1019.017,338.012,355.102,170.940,50.245,159.871
C07931=1019.011,337.765,355.137,170.933,50.248,159.870
C07932=1019.003,337.513,355.174,170.926,50.251,159.870
C07933=1018.995,337.262,355.210,170.919,50.253,159.869
C07934=1018.989,337.010,355.246,170.912,50.256,159.869
C07935=1018.981,336.759,355.282,170.905,50.259,159.868
C07936=1018.974,336.512,355.317,170.899,50.261,159.868
C07937=1018.967,336.265,355.353,170.892,50.264,159.867
C07938=1018.960,336.017,355.389,170.885,50.267,159.867
C07939=1018.953,335.770,355.424,170.878,50.269,159.866
C07940=1018.946,335.523,355.460,170.871,50.272,159.866
C07941=1018.938,335.275,355.495,170.864,50.274,159.865
C07942=1018.932,335.027,355.530,170.858,50.277,159.865
C07943=1018.925,334.780,355.565,170.851,50.280,159.864
C07944=1018.917,334.533,355.602,170.844,50.283,159.864
C07945=1018.910,334.285,355.637,170.837,50.285,159.863
C07946=1018.904,334.038,355.672,170.830,50.288,159.863
C07947=1018.897,333.790,355.707,170.823,50.291,159.862
C07948=1018.890,333.542,355.742,170.817,50.294,159.862
C07949=1018.882,333.296,355.778,170.810,50.297,159.861
C07950=1018.876,333.048,355.813,170.803,50.299,159.861
C07951=1018.869,332.801,355.849,170.797,50.302,159.860
C07952=1018.861,332.554,355.883,170.789,50.305,159.860
C07953=1018.854,332.306,355.919,170.783,50.308,159.859
C07954=1018.847,332.058,355.954,170.776,50.311,159.859
C07955=1018.841,331.811,355.989,170.770,50.314,159.859
C07956=1018.833,331.564,356.023,170.763,50.317,159.858
C07957=1018.826,331.317,356.059,170.757,50.319,159.858
C07958=1018.820,331.069,356.093,170.750,50.322,159.857
C07959=1018.812,330.821,356.128,170.744,50.325,159.857
C07960=1018.805,330.574,356.163,170.737,50.328,159.857
C07961=1018.798,330.326,356.198,170.730,50.331,159.856
C07962=1018.791,330.079,356.233,170.724,50.334,159.856
C07963=1018.784,329.831,356.267,170.717,50.337,159.855
C07964=1018.777,329.584,356.302,170.710,50.340,159.855
C07965=1018.771,329.336,356.337,170.703,50.343,159.854
C07966=1018.763,329.089,356.372,170.697,50.346,159.854
C07967=1018.757,328.841,356.406,170.690,50.349,159.854
C07968=1018.750,328.594,356.442,170.684,50.352,159.853
C07969=1018.743,328.347,356.477,170.678,50.355,159.853
C07970=1018.736,328.099,356.510,170.671,50.358,159.852
C07971=1018.729,327.852,356.546,170.665,50.361,159.852
C07972=1018.723,327.604,356.580,170.658,50.364,159.852
C07973=1018.715,327.357,356.615,170.651,50.367,159.851
C07974=1018.708,327.109,356.650,170.645,50.371,159.851
C07975=1018.702,326.861,356.684,170.638,50.374,159.851
C07976=1018.694,326.614,356.719,170.632,50.377,159.850
C07977=1018.688,326.366,356.753,170.626,50.379,159.850
C07978=1018.681,326.119,356.787,170.620,50.383,159.850
C07979=1018.675,325.872,356.822,170.613,50.386,159.849
C07980=1018.667,325.624,356.855,170.607,50.389,159.849
C07981=1018.660,325.377,356.889,170.600,50.392,159.849
C07982=1018.653,325.129,356.923,170.593,50.395,159.848
C07983=1018.646,324.881,356.958,170.587,50.399,159.848
C07984=1018.639,324.634,356.992,170.581,50.402,159.848
C07985=1018.632,324.386,357.026,170.574,50.406,159.847
C07986=1018.625,324.138,357.060,170.568,50.409,159.847
C07987=1018.618,323.890,357.094,170.561,50.412,159.847
C07988=1018.612,323.643,357.128,170.555,50.416,159.846
C07989=1018.604,323.396,357.161,170.548,50.419,159.846
C07990=1018.598,323.148,357.197,170.543,50.422,159.846
C07991=1018.590,322.901,357.230,170.536,50.425,159.846
C07992=1018.583,322.645,357.265,170.529,50.429,159.845
C07993=1018.576,322.389,357.300,170.522,50.432,159.845
C07994=1018.569,322.134,357.335,170.516,50.436,159.845
C07995=1018.562,321.878,357.370,170.510,50.440,159.844
C07996=1018.555,321.631,357.404,170.503,50.443,159.844
C07997=1018.548,321.383,357.438,170.497,50.447,159.844
C07998=1018.542,321.136,357.472,170.490,50.450,159.843
C07999=1018.535,320.887,357.505,170.485,50.453,159.843
C08000=1018.528,320.640,357.539,170.479,50.457,159.843
C08001=1018.521,320.392,357.573,170.472,50.460,159.843
C08002=1018.515,320.145,357.607,170.466,50.463,159.843
C08003=1018.507,319.897,357.640,170.460,50.467,159.842
C08004=1018.501,319.650,357.674,170.453,50.470,159.842
C08005=1018.494,319.402,357.707,170.447,50.474,159.842
C08006=1018.488,319.154,357.741,170.442,50.477,159.842
C08007=1018.481,318.907,357.775,170.435,50.480,159.841
C08008=1018.474,318.659,357.809,170.429,50.484,159.841
C08009=1018.467,318.411,357.843,170.422,50.488,159.841
C08010=1018.461,318.164,357.876,170.416,50.492,159.841
C08011=1018.454,317.916,357.910,170.409,50.495,159.840
C08012=1018.447,317.669,357.943,170.404,50.498,159.840
C08013=1018.440,317.421,357.976,170.398,50.502,159.840
C08014=1018.434,317.173,358.010,170.392,50.505,159.840
C08015=1018.427,316.926,358.044,170.386,50.509,159.840
C08016=1018.421,316.678,358.077,170.379,50.513,159.839
C08017=1018.414,316.430,358.111,170.373,50.517,159.839
C08018=1018.408,316.182,358.144,170.367,50.519,159.839
C08019=1018.401,315.935,358.178,170.361,50.523,159.839
C08020=1018.395,315.687,358.211,170.355,50.527,159.838
C08021=1018.387,315.439,358.244,170.349,50.530,159.838
C08022=1018.381,315.192,358.277,170.342,50.534,159.838
C08023=1018.375,314.945,358.311,170.337,50.537,159.838
C08024=1018.368,314.696,358.344,170.331,50.541,159.838
C08025=1018.362,314.449,358.378,170.325,50.545,159.837
C08026=1018.355,314.201,358.411,170.318,50.549,159.837
C08027=1018.349,313.954,358.445,170.312,50.552,159.837
C08028=1018.343,313.706,358.478,170.307,50.556,159.837
C08029=1018.336,313.459,358.512,170.301,50.559,159.837
C08030=1018.329,313.211,358.544,170.294,50.563,159.837
C08031=1018.323,312.963,358.577,170.289,50.568,159.837
C08032=1018.317,312.715,358.611,170.282,50.571,159.836
C08033=1018.310,312.468,358.644,170.277,50.575,159.836
C08034=1018.304,312.220,358.677,170.271,50.578,159.836
C08035=1018.297,311.973,358.710,170.265,50.582,159.836
C08036=1018.290,311.725,358.743,170.258,50.586,159.836
C08037=1018.285,311.477,358.777,170.253,50.589,159.835
C08038=1018.279,311.229,358.810,170.247,50.594,159.835
C08039=1018.272,310.982,358.843,170.241,50.597,159.835
C08040=1018.265,310.734,358.876,170.235,50.601,159.835
C08041=1018.260,310.486,358.909,170.229,50.604,159.835
C08042=1018.253,310.239,358.942,170.223,50.608,159.835
C08043=1018.247,309.991,358.975,170.217,50.613,159.835
C08044=1018.241,309.743,359.008,170.211,50.616,159.835
C08045=1018.234,309.496,359.040,170.206,50.620,159.834
C08046=1018.227,309.248,359.073,170.200,50.624,159.834
C08047=1018.220,309.000,359.106,170.194,50.628,159.834
C08048=1018.213,308.753,359.138,170.188,50.632,159.834
C08049=1018.207,308.505,359.171,170.182,50.637,159.834
C08050=1018.201,308.257,359.203,170.176,50.640,159.834
C08051=1018.194,308.009,359.235,170.170,50.645,159.834
C08052=1018.187,307.759,359.268,170.164,50.648,159.834
C08053=1018.180,307.509,359.301,170.158,50.653,159.834
C08054=1018.174,307.258,359.333,170.153,50.657,159.834
C08055=1018.167,307.009,359.366,170.147,50.661,159.834
C08056=1018.161,306.761,359.398,170.141,50.665,159.834
C08057=1018.153,306.513,359.430,170.135,50.669,159.834
C08058=1018.147,306.265,359.463,170.129,50.673,159.833
C08059=1018.141,306.017,359.495,170.123,50.677,159.833
C08060=1018.134,305.769,359.527,170.117,50.682,159.833
C08061=1018.128,305.521,359.559,170.112,50.686,159.834
C08062=1018.121,305.274,359.592,170.106,50.690,159.833
C08063=1018.115,305.026,359.624,170.100,50.694,159.833
C08064=1018.108,304.778,359.656,170.094,50.698,159.833
C08065=1018.102,304.531,359.688,170.088,50.703,159.833
C08066=1018.096,304.283,359.721,170.082,50.707,159.833
C08067=1018.089,304.035,359.753,170.077,50.711,159.833
C08068=1018.083,303.787,359.785,170.071,50.715,159.833
C08069=1018.076,303.539,359.816,170.066,50.719,159.833
C08070=1018.070,303.292,359.849,170.060,50.724,159.833
C08071=1018.063,303.044,359.880,170.054,50.728,159.833
C08072=1018.057,302.796,359.913,170.048,50.732,159.833
C08073=1018.051,302.548,359.945,170.043,50.736,159.833
C08074=1018.044,302.300,359.976,170.037,50.740,159.833
C08075=1018.038,302.052,360.009,170.031,50.745,159.833
C08076=1018.031,301.805,360.041,170.025,50.749,159.833
C08077=1018.025,301.556,360.073,170.019,50.754,159.833
C08078=1018.018,301.309,360.105,170.015,50.758,159.833
C08079=1018.012,301.061,360.137,170.009,50.762,159.833
C08080=1018.005,300.813,360.168,170.003,50.766,159.833
C08081=1017.999,300.565,360.201,169.997,50.771,159.833
C08082=1017.993,300.317,360.233,169.991,50.775,159.833
C08083=1017.987,300.070,360.264,169.986,50.779,159.833
C08084=1017.981,299.822,360.296,169.980,50.784,159.833
C08085=1017.974,299.574,360.328,169.975,50.788,159.833
C08086=1017.968,299.326,360.360,169.969,50.792,159.833
C08087=1017.961,299.078,360.392,169.963,50.797,159.833
C08088=1017.955,298.830,360.424,169.958,50.801,159.833
C08089=1017.949,298.583,360.455,169.953,50.806,159.833
C08090=1017.943,298.335,360.487,169.947,50.810,159.833
C08091=1017.937,298.086,360.519,169.941,50.815,159.833
C08092=1017.930,297.839,360.550,169.936,50.819,159.833
C08093=1017.924,297.590,360.582,169.930,50.823,159.833
C08094=1017.918,297.344,360.614,169.924,50.828,159.833
C08095=1017.912,297.096,360.646,169.919,50.833,159.834
C08096=1017.905,296.848,360.678,169.913,50.837,159.834
C08097=1017.899,296.599,360.710,169.908,50.841,159.834
C08098=1017.893,296.352,360.741,169.902,50.846,159.834
C08099=1017.887,296.104,360.773,169.896,50.850,159.834
C08100=1017.881,295.856,360.805,169.891,50.855,159.834
C08101=1017.875,295.608,360.835,169.886,50.859,159.834
C08102=1017.869,295.360,360.867,169.880,50.864,159.834
C08103=1017.862,295.112,360.899,169.875,50.869,159.834
C08104=1017.857,294.864,360.930,169.869,50.873,159.834
C08105=1017.850,294.616,360.962,169.863,50.878,159.834
C08106=1017.844,294.368,360.994,169.859,50.882,159.834
C08107=1017.838,294.121,361.025,169.853,50.887,159.834
C08108=1017.832,293.881,361.056,169.847,50.891,159.834
C08109=1017.827,293.640,361.087,169.842,50.895,159.834
C08110=1017.821,293.400,361.116,169.837,50.900,159.835
C08111=1017.815,293.160,361.147,169.832,50.904,159.835
C08112=1017.809,292.919,361.178,169.826,50.909,159.835
C08113=1017.803,292.680,361.208,169.822,50.913,159.835
C08114=1017.797,292.439,361.238,169.816,50.918,159.835
C08115=1017.791,292.199,361.267,169.810,50.923,159.835
C08116=1017.785,291.951,361.299,169.806,50.927,159.835
C08117=1017.778,291.703,361.331,169.800,50.932,159.835
C08118=1017.772,291.455,361.361,169.795,50.937,159.836
C08119=1017.766,291.207,361.392,169.789,50.942,159.836
C08120=1017.760,290.960,361.423,169.783,50.947,159.836
C08121=1017.753,290.712,361.454,169.778,50.952,159.836
C08122=1017.748,290.464,361.485,169.773,50.956,159.836
C08123=1017.742,290.215,361.516,169.768,50.961,159.836
C08124=1017.736,289.968,361.547,169.762,50.966,159.836
C08125=1017.729,289.719,361.578,169.757,50.971,159.837
C08126=1017.723,289.472,361.609,169.751,50.976,159.837
C08127=1017.717,289.224,361.639,169.745,50.981,159.837
C08128=1017.710,288.975,361.670,169.740,50.986,159.837
C08129=1017.704,288.728,361.701,169.736,50.991,159.837
C08130=1017.698,288.479,361.732,169.730,50.995,159.837
C08131=1017.692,288.232,361.762,169.724,51.000,159.838
C08132=1017.686,287.984,361.793,169.719,51.005,159.838
C08133=1017.679,287.736,361.824,169.713,51.010,159.838
C08134=1017.673,287.488,361.854,169.708,51.015,159.838
C08135=1017.667,287.239,361.885,169.704,51.020,159.838
C08136=1017.661,286.992,361.915,169.698,51.025,159.839
C08137=1017.655,286.743,361.946,169.693,51.030,159.839
C08138=1017.649,286.496,361.977,169.687,51.035,159.839
C08139=1017.642,286.247,362.008,169.682,51.040,159.839
C08140=1017.636,286.000,362.038,169.676,51.046,159.839
C08141=1017.631,285.752,362.069,169.671,51.051,159.840
C08142=1017.624,285.503,362.099,169.666,51.055,159.840
C08143=1017.618,285.255,362.130,169.661,51.061,159.840
C08144=1017.612,285.007,362.160,169.656,51.066,159.840
C08145=1017.606,284.759,362.191,169.650,51.071,159.840
C08146=1017.600,284.511,362.221,169.645,51.076,159.841
C08147=1017.594,284.263,362.252,169.639,51.081,159.841
C08148=1017.587,284.015,362.282,169.634,51.086,159.841
C08149=1017.582,283.767,362.312,169.629,51.091,159.841
C08150=1017.575,283.519,362.343,169.624,51.096,159.841
C08151=1017.569,283.271,362.373,169.619,51.102,159.842
C08152=1017.563,283.024,362.403,169.614,51.107,159.842
C08153=1017.557,282.774,362.433,169.608,51.112,159.842
C08154=1017.551,282.527,362.463,169.603,51.117,159.842
C08155=1017.545,282.279,362.493,169.597,51.122,159.843
C08156=1017.538,282.031,362.524,169.592,51.128,159.843
C08157=1017.532,281.783,362.554,169.587,51.133,159.843
C08158=1017.527,281.534,362.584,169.582,51.138,159.843
C08159=1017.521,281.286,362.614,169.577,51.144,159.844
C08160=1017.514,281.038,362.644,169.572,51.149,159.844
C08161=1017.508,280.790,362.674,169.566,51.154,159.844
C08162=1017.502,280.542,362.704,169.561,51.160,159.845
C08163=1017.496,280.294,362.734,169.556,51.165,159.845
C08164=1017.489,280.046,362.764,169.551,51.170,159.845
C08165=1017.484,279.798,362.794,169.546,51.176,159.845
C08166=1017.478,279.550,362.824,169.540,51.181,159.846
C08167=1017.472,279.302,362.855,169.536,51.186,159.846
C08168=1017.466,279.067,362.883,169.531,51.191,159.846
C08169=1017.461,278.833,362.911,169.526,51.196,159.846
C08170=1017.455,278.600,362.939,169.521,51.201,159.847
C08171=1017.449,278.365,362.968,169.516,51.206,159.847
C08172=1017.443,278.131,362.995,169.511,51.211,159.847
C08173=1017.438,277.897,363.024,169.507,51.217,159.848
C08174=1017.433,277.663,363.053,169.501,51.222,159.848
C08175=1017.427,277.429,363.080,169.497,51.226,159.848
C08176=1017.421,277.181,363.111,169.492,51.232,159.848
C08177=1017.415,276.933,363.140,169.487,51.237,159.849
C08178=1017.409,276.685,363.170,169.482,51.243,159.849
C08179=1017.403,276.437,363.200,169.476,51.248,159.849
C08180=1017.397,276.188,363.230,169.471,51.254,159.850
C08181=1017.391,275.940,363.259,169.466,51.259,159.850
C08182=1017.385,275.692,363.289,169.461,51.265,159.850
C08183=1017.379,275.444,363.319,169.456,51.271,159.851
C08184=1017.372,275.196,363.348,169.451,51.277,159.851
C08185=1017.367,274.947,363.378,169.445,51.282,159.851
C08186=1017.360,274.700,363.407,169.440,51.288,159.852
C08187=1017.355,274.452,363.437,169.436,51.293,159.852
C08188=1017.349,274.203,363.466,169.431,51.298,159.852
C08189=1017.343,273.955,363.496,169.426,51.304,159.853
C08190=1017.336,273.707,363.525,169.421,51.310,159.853
C08191=1017.331,273.459,363.555,169.416,51.316,159.853
C08192=1017.325,273.211,363.584,169.411,51.321,159.854
C08193=1017.319,272.962,363.614,169.405,51.327,159.854
C08194=1017.313,272.714,363.643,169.400,51.332,159.854
C08195=1017.307,272.466,363.673,169.395,51.338,159.855
C08196=1017.301,272.218,363.702,169.390,51.344,159.855
C08197=1017.295,271.970,363.732,169.385,51.350,159.856
C08198=1017.289,271.722,363.761,169.380,51.356,159.856
C08199=1017.283,271.474,363.790,169.375,51.361,159.856
C08200=1017.277,271.225,363.819,169.370,51.367,159.856
C08201=1017.271,270.977,363.848,169.365,51.372,159.857
C08202=1017.266,270.729,363.878,169.360,51.378,159.857
C08203=1017.259,270.480,363.907,169.355,51.384,159.858
C08204=1017.253,270.232,363.936,169.350,51.390,159.858
C08205=1017.248,269.984,363.966,169.345,51.396,159.858
C08206=1017.241,269.736,363.995,169.340,51.402,159.859
C08207=1017.236,269.487,364.025,169.335,51.407,159.859
C08208=1017.230,269.239,364.054,169.330,51.413,159.860
C08209=1017.224,268.992,364.082,169.325,51.419,159.860
C08210=1017.218,268.743,364.112,169.320,51.426,159.861
C08211=1017.212,268.495,364.141,169.315,51.431,159.861
C08212=1017.206,268.246,364.169,169.310,51.437,159.861
C08213=1017.200,267.998,364.198,169.305,51.443,159.862
C08214=1017.194,267.750,364.227,169.300,51.449,159.862
C08215=1017.188,267.502,364.257,169.295,51.455,159.863
C08216=1017.183,267.254,364.286,169.290,51.461,159.863
C08217=1017.177,267.006,364.314,169.286,51.467,159.863
C08218=1017.170,266.757,364.343,169.281,51.473,159.864
C08219=1017.165,266.509,364.373,169.276,51.479,159.864
C08220=1017.159,266.260,364.401,169.271,51.485,159.865
C08221=1017.153,266.012,364.430,169.266,51.491,159.865
C08222=1017.147,265.765,364.459,169.261,51.497,159.866
C08223=1017.141,265.517,364.488,169.256,51.503,159.866
C08224=1017.136,265.267,364.517,169.251,51.509,159.866
C08225=1017.129,265.019,364.546,169.247,51.515,159.867
C08226=1017.123,264.771,364.574,169.242,51.521,159.867
C08227=1017.118,264.523,364.603,169.237,51.527,159.868
C08228=1017.112,264.291,364.629,169.233,51.532,159.868
C08229=1017.106,264.059,364.657,169.228,51.539,159.869
C08230=1017.101,263.827,364.683,169.223,51.545,159.869
C08231=1017.095,263.595,364.709,169.219,51.550,159.870
C08232=1017.090,263.364,364.737,169.214,51.556,159.870
C08233=1017.084,263.132,364.763,169.210,51.561,159.871
C08234=1017.079,262.900,364.789,169.205,51.567,159.871
C08235=1017.073,262.669,364.817,169.200,51.573,159.871
C08236=1017.067,262.420,364.845,169.195,51.579,159.872
C08237=1017.061,262.172,364.874,169.191,51.586,159.872
C08238=1017.056,261.924,364.902,169.186,51.591,159.873
C08239=1017.050,261.675,364.930,169.181,51.598,159.873
C08240=1017.044,261.427,364.959,169.176,51.604,159.874
C08241=1017.038,261.179,364.987,169.171,51.610,159.874
C08242=1017.032,260.931,365.016,169.167,51.617,159.875
C08243=1017.027,260.682,365.045,169.162,51.623,159.875
C08244=1017.021,260.434,365.073,169.157,51.629,159.876
C08245=1017.015,260.185,365.102,169.152,51.635,159.876
C08246=1017.009,259.937,365.130,169.148,51.642,159.877
C08247=1017.004,259.689,365.158,169.143,51.648,159.877
C08248=1016.997,259.440,365.186,169.137,51.654,159.878
C08249=1016.991,259.191,365.215,169.133,51.661,159.878
C08250=1016.986,258.943,365.242,169.128,51.667,159.879
C08251=1016.979,258.696,365.271,169.124,51.674,159.880
C08252=1016.973,258.447,365.299,169.119,51.681,159.880
C08253=1016.967,258.199,365.327,169.114,51.687,159.881
C08254=1016.961,257.950,365.355,169.108,51.693,159.881
C08255=1016.955,257.702,365.383,169.104,51.700,159.882
C08256=1016.949,257.454,365.411,169.099,51.706,159.882
C08257=1016.943,257.205,365.439,169.095,51.713,159.883
C08258=1016.938,256.957,365.467,169.090,51.720,159.883
C08259=1016.931,256.709,365.495,169.085,51.726,159.884
C08260=1016.925,256.460,365.523,169.080,51.733,159.884
C08261=1016.919,256.212,365.550,169.076,51.740,159.885
C08262=1016.913,255.963,365.578,169.071,51.746,159.886
C08263=1016.908,255.715,365.606,169.066,51.753,159.886
C08264=1016.901,255.466,365.634,169.061,51.760,159.887
C08265=1016.896,255.218,365.662,169.056,51.766,159.887
C08266=1016.890,254.969,365.690,169.052,51.773,159.888
C08267=1016.884,254.722,365.717,169.047,51.779,159.889
C08268=1016.878,254.473,365.746,169.043,51.786,159.889
C08269=1016.872,254.224,365.774,169.037,51.793,159.890
C08270=1016.866,253.976,365.801,169.033,51.799,159.890
C08271=1016.860,253.727,365.829,169.028,51.806,159.891
C08272=1016.854,253.479,365.856,169.023,51.812,159.891
C08273=1016.849,253.231,365.884,169.019,51.819,159.892
C08274=1016.843,252.982,365.913,169.013,51.826,159.893
C08275=1016.837,252.735,365.940,169.009,51.832,159.893
C08276=1016.831,252.485,365.968,169.004,51.839,159.894
C08277=1016.826,252.237,365.995,169.000,51.846,159.894
C08278=1016.819,251.989,366.023,168.996,51.853,159.895
C08279=1016.814,251.741,366.051,168.990,51.860,159.896
C08280=1016.808,251.492,366.078,168.986,51.866,159.896
C08281=1016.802,251.244,366.106,168.981,51.873,159.897
C08282=1016.797,250.996,366.134,168.976,51.879,159.897
C08283=1016.790,250.747,366.161,168.971,51.887,159.898
C08284=1016.785,250.499,366.189,168.967,51.894,159.899
C08285=1016.778,250.250,366.217,168.962,51.900,159.899
C08286=1016.773,250.001,366.244,168.958,51.907,159.900
C08287=1016.768,249.753,366.272,168.952,51.914,159.900
C08288=1016.762,249.520,366.298,168.949,51.920,159.901
C08289=1016.757,249.288,366.323,168.944,51.927,159.902
C08290=1016.752,249.055,366.349,168.940,51.933,159.902
C08291=1016.747,248.823,366.375,168.935,51.940,159.903
C08292=1016.741,248.590,366.401,168.932,51.946,159.904
C08293=1016.736,248.357,366.427,168.927,51.953,159.904
C08294=1016.730,248.125,366.453,168.923,51.959,159.905
C08295=1016.725,247.891,366.479,168.918,51.966,159.905
C08296=1016.719,247.643,366.506,168.913,51.972,159.906
C08297=1016.714,247.395,366.534,168.909,51.979,159.906
C08298=1016.708,247.147,366.560,168.905,51.986,159.907
C08299=1016.702,246.898,366.588,168.899,51.993,159.908
C08300=1016.697,246.649,366.616,168.895,52.000,159.909
C08301=1016.691,246.402,366.643,168.891,52.007,159.909
C08302=1016.686,246.153,366.670,168.886,52.014,159.910
C08303=1016.680,245.904,366.699,168.881,52.021,159.910
C08304=1016.674,245.656,366.725,168.877,52.028,159.911
C08305=1016.669,245.408,366.753,168.872,52.035,159.912
C08306=1016.663,245.159,366.780,168.867,52.042,159.912
C08307=1016.657,244.910,366.808,168.863,52.049,159.913
C08308=1016.652,244.662,366.835,168.858,52.056,159.914
C08309=1016.646,244.414,366.862,168.854,52.063,159.915
C08310=1016.641,244.166,366.890,168.849,52.070,159.915
C08311=1016.635,243.917,366.917,168.845,52.078,159.916
C08312=1016.630,243.668,366.944,168.840,52.084,159.916
C08313=1016.624,243.420,366.972,168.836,52.091,159.917
C08314=1016.618,243.171,366.999,168.831,52.098,159.918
C08315=1016.613,242.923,367.026,168.826,52.106,159.919
C08316=1016.607,242.675,367.054,168.822,52.113,159.919
C08317=1016.601,242.426,367.081,168.817,52.120,159.920
C08318=1016.596,242.177,367.108,168.813,52.127,159.921
C08319=1016.590,241.929,367.134,168.809,52.135,159.921
C08320=1016.584,241.681,367.161,168.803,52.142,159.922
C08321=1016.579,241.432,367.188,168.799,52.149,159.923
C08322=1016.574,241.183,367.215,168.794,52.157,159.923
C08323=1016.567,240.934,367.242,168.790,52.164,159.924
C08324=1016.562,240.686,367.270,168.786,52.171,159.925
C08325=1016.556,240.438,367.297,168.780,52.178,159.926
C08326=1016.550,240.190,367.323,168.776,52.185,159.926
C08327=1016.545,239.941,367.351,168.772,52.193,159.927
C08328=1016.539,239.693,367.377,168.767,52.200,159.928
C08329=1016.534,239.444,367.404,168.763,52.208,159.929
C08330=1016.528,239.196,367.430,168.758,52.215,159.929
C08331=1016.523,238.947,367.458,168.754,52.222,159.930
C08332=1016.517,238.699,367.484,168.750,52.229,159.931
C08333=1016.511,238.451,367.511,168.744,52.237,159.931
C08334=1016.506,238.202,367.538,168.740,52.244,159.932
C08335=1016.500,237.954,367.564,168.735,52.252,159.933
C08336=1016.494,237.704,367.591,168.731,52.259,159.934
C08337=1016.488,237.456,367.617,168.726,52.267,159.934
C08338=1016.482,237.207,367.644,168.723,52.275,159.936
C08339=1016.476,236.959,367.671,168.718,52.283,159.936
C08340=1016.471,236.711,367.697,168.713,52.290,159.937
C08341=1016.465,236.462,367.723,168.708,52.298,159.938
C08342=1016.459,236.213,367.750,168.704,52.305,159.939
C08343=1016.454,235.965,367.776,168.699,52.313,159.939
C08344=1016.448,235.717,367.803,168.695,52.320,159.940
C08345=1016.442,235.468,367.829,168.690,52.328,159.941
C08346=1016.437,235.219,367.856,168.687,52.336,159.942
C08347=1016.431,234.971,367.882,168.682,52.344,159.942
C08348=1016.426,234.735,367.907,168.677,52.351,159.943
C08349=1016.420,234.499,367.933,168.673,52.358,159.944
C08350=1016.415,234.263,367.957,168.669,52.365,159.945
C08351=1016.410,234.027,367.982,168.665,52.372,159.945
C08352=1016.404,233.791,368.007,168.661,52.380,159.946
C08353=1016.399,233.555,368.033,168.656,52.387,159.947
C08354=1016.393,233.318,368.057,168.652,52.395,159.948
C08355=1016.388,233.082,368.082,168.648,52.402,159.949
C08356=1016.383,232.834,368.109,168.643,52.410,159.949
C08357=1016.377,232.586,368.136,168.639,52.417,159.950
C08358=1016.371,232.337,368.162,168.634,52.425,159.951
C08359=1016.366,232.088,368.188,168.630,52.433,159.952
C08360=1016.360,231.839,368.214,168.625,52.440,159.953
C08361=1016.354,231.591,368.241,168.621,52.448,159.954
C08362=1016.349,231.342,368.267,168.616,52.456,159.954
C08363=1016.344,231.094,368.293,168.613,52.464,159.955
C08364=1016.338,230.845,368.319,168.608,52.472,159.956
C08365=1016.332,230.597,368.345,168.603,52.480,159.957
C08366=1016.326,230.348,368.371,168.599,52.488,159.958
C08367=1016.321,230.100,368.398,168.594,52.495,159.958
C08368=1016.315,229.851,368.423,168.591,52.504,159.959
C08369=1016.309,229.602,368.450,168.585,52.511,159.960
C08370=1016.304,229.354,368.476,168.581,52.520,159.961
C08371=1016.299,229.106,368.502,168.577,52.527,159.962
C08372=1016.293,228.857,368.528,168.572,52.535,159.963
C08373=1016.287,228.608,368.554,168.568,52.543,159.964
C08374=1016.281,228.360,368.580,168.564,52.551,159.965
C08375=1016.276,228.111,368.606,168.559,52.559,159.965
C08376=1016.271,227.863,368.632,168.555,52.567,159.966
C08377=1016.265,227.614,368.658,168.551,52.575,159.967
C08378=1016.259,227.366,368.684,168.546,52.583,159.968
C08379=1016.253,227.117,368.710,168.542,52.591,159.969
C08380=1016.248,226.868,368.736,168.537,52.600,159.970
C08381=1016.243,226.620,368.762,168.532,52.607,159.970
C08382=1016.237,226.371,368.788,168.529,52.616,159.972
C08383=1016.231,226.122,368.813,168.524,52.624,159.972
C08384=1016.226,225.873,368.839,168.519,52.632,159.973
C08385=1016.220,225.625,368.864,168.516,52.640,159.974
C08386=1016.215,225.376,368.890,168.511,52.648,159.975
C08387=1016.209,225.127,368.916,168.507,52.657,159.976
C08388=1016.203,224.879,368.941,168.502,52.665,159.977
C08389=1016.198,224.630,368.967,168.497,52.674,159.978
C08390=1016.192,224.382,368.993,168.493,52.681,159.979
C08391=1016.186,224.133,369.019,168.489,52.689,159.980
C08392=1016.180,223.885,369.044,168.484,52.698,159.981
C08393=1016.175,223.636,369.070,168.480,52.706,159.981
C08394=1016.169,223.388,369.095,168.476,52.714,159.982
C08395=1016.163,223.139,369.121,168.472,52.723,159.983
C08396=1016.158,222.890,369.147,168.467,52.731,159.984
C08397=1016.152,222.642,369.172,168.463,52.740,159.985
C08398=1016.147,222.393,369.198,168.458,52.748,159.986
C08399=1016.141,222.144,369.222,168.454,52.756,159.987
C08400=1016.136,221.895,369.248,168.450,52.765,159.988
C08401=1016.130,221.647,369.273,168.445,52.773,159.989
C08402=1016.124,221.398,369.299,168.441,52.782,159.990
C08403=1016.119,221.150,369.324,168.436,52.790,159.991
C08404=1016.113,220.901,369.350,168.433,52.798,159.992
C08405=1016.108,220.652,369.376,168.428,52.807,159.993
C08406=1016.102,220.404,369.401,168.424,52.815,159.994
C08407=1016.097,220.155,369.427,168.419,52.824,159.995
C08408=1016.091,219.915,369.451,168.416,52.832,159.996
C08409=1016.086,219.675,369.476,168.411,52.840,159.997
C08410=1016.081,219.434,369.500,168.406,52.848,159.997
C08411=1016.075,219.194,369.525,168.403,52.856,159.998
C08412=1016.070,218.954,369.549,168.398,52.865,159.999
C08413=1016.065,218.714,369.574,168.395,52.873,160.000
C08414=1016.059,218.473,369.598,168.390,52.881,160.001
C08415=1016.054,218.233,369.623,168.387,52.889,160.002
C08416=1016.048,217.984,369.648,168.382,52.898,160.003
C08417=1016.043,217.736,369.673,168.378,52.906,160.004
C08418=1016.037,217.487,369.699,168.373,52.916,160.005
C08419=1016.032,217.239,369.723,168.369,52.924,160.006
C08420=1016.026,216.990,369.749,168.364,52.933,160.007
C08421=1016.020,216.741,369.773,168.360,52.942,160.008
C08422=1016.015,216.492,369.799,168.356,52.950,160.009
C08423=1016.009,216.244,369.824,168.351,52.959,160.010
C08424=1016.003,215.995,369.848,168.347,52.968,160.011
C08425=1015.997,215.746,369.874,168.343,52.976,160.012
C08426=1015.993,215.498,369.899,168.339,52.986,160.013
C08427=1015.986,215.249,369.924,168.334,52.994,160.014
C08428=1015.981,215.000,369.948,168.330,53.003,160.015
C08429=1015.975,214.752,369.973,168.326,53.012,160.016
C08430=1015.970,214.503,369.998,168.321,53.020,160.017
C08431=1015.964,214.254,370.024,168.317,53.030,160.018
C08432=1015.959,214.006,370.048,168.313,53.038,160.019
C08433=1015.953,213.757,370.073,168.309,53.047,160.020
C08434=1015.948,213.508,370.098,168.304,53.056,160.021
C08435=1015.942,213.259,370.123,168.300,53.065,160.023
C08436=1015.937,213.011,370.148,168.296,53.074,160.023
C08437=1015.931,212.763,370.173,168.292,53.083,160.025
C08438=1015.926,212.513,370.198,168.287,53.092,160.026
C08439=1015.920,212.265,370.223,168.283,53.100,160.027
C08440=1015.914,212.016,370.247,168.279,53.110,160.028
C08441=1015.909,211.767,370.272,168.274,53.118,160.029
C08442=1015.904,211.518,370.298,168.270,53.127,160.030
C08443=1015.898,211.270,370.322,168.266,53.137,160.031
C08444=1015.893,211.022,370.347,168.262,53.145,160.032
C08445=1015.887,210.772,370.371,168.258,53.154,160.033
C08446=1015.881,210.524,370.396,168.254,53.164,160.034
C08447=1015.876,210.275,370.422,168.249,53.172,160.035
C08448=1015.871,210.026,370.446,168.244,53.182,160.036
C08449=1015.865,209.778,370.470,168.240,53.191,160.037
C08450=1015.859,209.529,370.496,168.236,53.200,160.038
C08451=1015.854,209.280,370.520,168.232,53.209,160.039
C08452=1015.849,209.032,370.544,168.228,53.218,160.041
C08453=1015.843,208.782,370.569,168.224,53.227,160.042
C08454=1015.838,208.534,370.594,168.220,53.237,160.043
C08455=1015.832,208.285,370.619,168.215,53.245,160.044
C08456=1015.827,208.036,370.643,168.210,53.255,160.045
C08457=1015.821,207.788,370.667,168.206,53.264,160.046
C08458=1015.815,207.539,370.692,168.202,53.273,160.047
C08459=1015.810,207.290,370.716,168.198,53.283,160.048
C08460=1015.805,207.041,370.741,168.195,53.292,160.050
C08461=1015.800,206.793,370.765,168.189,53.301,160.051
C08462=1015.793,206.544,370.790,168.186,53.311,160.052
C08463=1015.788,206.296,370.814,168.182,53.320,160.053
C08464=1015.783,206.047,370.839,168.178,53.329,160.054
C08465=1015.777,205.798,370.863,168.173,53.339,160.055
C08466=1015.772,205.549,370.887,168.169,53.348,160.056
C08467=1015.765,205.301,370.911,168.165,53.357,160.057
C08468=1015.760,205.064,370.935,168.160,53.366,160.058
C08469=1015.755,204.829,370.957,168.156,53.375,160.059
C08470=1015.750,204.593,370.980,168.152,53.384,160.061
C08471=1015.745,204.357,371.004,168.149,53.393,160.062
C08472=1015.739,204.121,371.027,168.145,53.402,160.063
C08473=1015.734,203.885,371.049,168.141,53.411,160.064
C08474=1015.729,203.650,371.072,168.137,53.421,160.065
C08475=1015.723,203.413,371.095,168.132,53.429,160.066
C08476=1015.701,202.198,371.205,167.622,53.370,159.946
C08477=1015.697,201.954,371.227,167.617,53.381,159.947
C08478=1015.693,201.711,371.250,167.611,53.391,159.948
C08479=1015.688,201.468,371.271,167.607,53.402,159.949
C08480=1015.684,201.218,371.294,167.602,53.412,159.950
C08481=1015.679,200.970,371.317,167.598,53.423,159.952
C08482=1015.674,200.721,371.339,167.593,53.434,159.953
C08483=1015.670,200.472,371.361,167.589,53.444,159.954
C08484=1015.666,200.223,371.383,167.584,53.455,159.955
C08485=1015.661,199.974,371.405,167.579,53.466,159.957
C08486=1015.657,199.725,371.429,167.574,53.476,159.958
C08487=1015.653,199.476,371.451,167.570,53.487,159.959
C08488=1015.648,199.227,371.473,167.566,53.498,159.960
C08489=1015.644,198.978,371.495,167.560,53.509,159.961
C08490=1015.639,198.729,371.518,167.556,53.520,159.963
C08491=1015.635,198.480,371.540,167.551,53.530,159.964
C08492=1015.630,198.231,371.562,167.546,53.541,159.965
C08493=1015.625,197.982,371.584,167.542,53.552,159.967
C08494=1015.620,197.733,371.606,167.537,53.562,159.968
C08495=1015.616,197.484,371.628,167.533,53.574,159.969
C08496=1015.611,197.235,371.650,167.527,53.584,159.970
C08497=1015.606,196.986,371.672,167.523,53.596,159.972
C08498=1015.602,196.737,371.694,167.519,53.606,159.973
C08499=1015.598,196.488,371.715,167.514,53.617,159.974
C08500=1015.593,196.239,371.737,167.509,53.628,159.975
C08501=1015.588,195.990,371.759,167.505,53.639,159.977
C08502=1015.584,195.741,371.782,167.501,53.650,159.978
C08503=1015.579,195.492,371.803,167.495,53.661,159.979
C08504=1015.574,195.243,371.825,167.491,53.671,159.980
C08505=1015.570,194.994,371.848,167.487,53.683,159.982
C08506=1015.566,194.745,371.869,167.482,53.693,159.983
C08507=1015.561,194.496,371.891,167.478,53.704,159.984
C08508=1015.556,194.247,371.913,167.473,53.715,159.986
C08509=1015.552,193.998,371.935,167.469,53.726,159.987
C08510=1015.547,193.749,371.957,167.464,53.737,159.988
C08511=1015.543,193.500,371.978,167.460,53.748,159.990
C08512=1015.539,193.251,372.001,167.455,53.758,159.991
C08513=1015.534,193.002,372.022,167.450,53.769,159.992
C08514=1015.529,192.753,372.044,167.446,53.780,159.993
C08515=1015.525,192.504,372.065,167.441,53.791,159.994
C08516=1015.520,192.230,372.089,167.437,53.803,159.996
C08517=1015.515,191.956,372.114,167.432,53.815,159.997
C08518=1015.511,191.683,372.138,167.427,53.827,159.999
C08519=1015.505,191.409,372.162,167.422,53.839,160.000
C08520=1015.501,191.160,372.183,167.418,53.850,160.002
C08521=1015.496,190.911,372.205,167.413,53.860,160.003
C08522=1015.493,190.662,372.227,167.408,53.872,160.004
C08523=1015.488,190.413,372.248,167.404,53.882,160.005
C08524=1015.483,190.164,372.270,167.400,53.893,160.007
C08525=1015.478,189.915,372.292,167.395,53.904,160.008
C08526=1015.475,189.665,372.314,167.391,53.915,160.009
C08527=1015.470,189.417,372.336,167.387,53.926,160.010
C08528=1015.466,189.168,372.356,167.383,53.937,160.012
C08529=1015.461,188.919,372.378,167.378,53.947,160.013
C08530=1015.457,188.670,372.401,167.374,53.959,160.014
C08531=1015.452,188.421,372.422,167.370,53.969,160.016
C08532=1015.448,188.172,372.444,167.365,53.980,160.017
C08533=1015.444,187.923,372.465,167.360,53.991,160.018
C08534=1015.440,187.674,372.487,167.356,54.002,160.019
C08535=1015.435,187.424,372.508,167.352,54.013,160.021
C08536=1015.430,187.145,372.533,167.347,54.025,160.022
C08537=1015.425,186.865,372.557,167.342,54.037,160.024
C08538=1015.421,186.585,372.581,167.338,54.049,160.025
C08539=1015.416,186.305,372.605,167.333,54.062,160.027
C08540=1015.412,186.057,372.627,167.329,54.072,160.028
C08541=1015.407,185.807,372.648,167.325,54.083,160.029
C08542=1015.402,185.559,372.670,167.320,54.094,160.031
C08543=1015.398,185.309,372.692,167.316,54.104,160.032
C08544=1015.394,185.061,372.713,167.312,54.116,160.033
C08545=1015.390,184.811,372.734,167.308,54.126,160.034
C08546=1015.386,184.562,372.757,167.304,54.137,160.036
C08547=1015.382,184.313,372.777,167.299,54.148,160.037
C08548=1015.377,184.065,372.799,167.295,54.159,160.038
C08549=1015.372,183.815,372.820,167.291,54.170,160.040
C08550=1015.369,183.566,372.842,167.286,54.180,160.041
C08551=1015.364,183.317,372.864,167.282,54.192,160.042
C08552=1015.360,183.068,372.885,167.278,54.202,160.043
C08553=1015.356,182.819,372.906,167.274,54.213,160.045
C08554=1015.352,182.570,372.928,167.270,54.224,160.046
C08555=1015.347,182.321,372.949,167.265,54.235,160.047
C08556=1015.343,182.072,372.970,167.261,54.246,160.049
C08557=1015.339,181.823,372.992,167.257,54.256,160.050
C08558=1015.335,181.573,373.014,167.253,54.268,160.051
C08559=1015.330,181.324,373.034,167.249,54.278,160.053
C08560=1015.326,181.075,373.055,167.245,54.290,160.054
C08561=1015.321,180.826,373.076,167.241,54.301,160.055
C08562=1015.316,180.577,373.097,167.237,54.312,160.057
C08563=1015.312,180.328,373.117,167.232,54.323,160.058
C08564=1015.307,180.079,373.138,167.229,54.334,160.059
C08565=1015.303,179.830,373.159,167.224,54.346,160.061
C08566=1015.298,179.581,373.180,167.220,54.357,160.062
C08567=1015.293,179.331,373.200,167.215,54.368,160.063
C08568=1015.289,179.082,373.220,167.211,54.379,160.065
C08569=1015.284,178.833,373.241,167.208,54.390,160.066
C08570=1015.280,178.584,373.262,167.204,54.402,160.068
C08571=1015.276,178.335,373.283,167.199,54.412,160.069
C08572=1015.270,178.086,373.304,167.195,54.423,160.070
C08573=1015.267,177.837,373.324,167.192,54.435,160.072
C08574=1015.261,177.588,373.345,167.187,54.445,160.073
C08575=1015.258,177.339,373.365,167.183,54.457,160.075
C08576=1015.253,177.089,373.386,167.179,54.468,160.076
C08577=1015.248,176.840,373.407,167.175,54.479,160.077
C08578=1015.244,176.591,373.427,167.170,54.490,160.078
C08579=1015.239,176.342,373.448,167.166,54.502,160.080
C08580=1015.235,176.094,373.469,167.162,54.513,160.081
C08581=1015.231,175.844,373.489,167.158,54.524,160.083
C08582=1015.226,175.595,373.509,167.154,54.535,160.084
C08583=1015.221,175.346,373.531,167.150,54.546,160.085
C08584=1015.217,175.097,373.551,167.146,54.557,160.087
C08585=1015.212,174.848,373.572,167.142,54.568,160.088
C08586=1015.209,174.599,373.592,167.138,54.580,160.090
C08587=1015.203,174.349,373.612,167.134,54.590,160.091
C08588=1015.199,174.101,373.633,167.130,54.602,160.092
C08589=1015.195,173.851,373.653,167.126,54.613,160.094
C08590=1015.191,173.602,373.674,167.122,54.624,160.095
C08591=1015.186,173.353,373.695,167.118,54.635,160.096
C08592=1015.181,173.104,373.715,167.114,54.646,160.098
C08593=1015.177,172.854,373.736,167.111,54.657,160.099
C08594=1015.173,172.606,373.756,167.107,54.668,160.101
C08595=1015.168,172.356,373.777,167.103,54.679,160.102
C08596=1015.164,172.107,373.797,167.099,54.690,160.103
C08597=1015.159,171.858,373.818,167.095,54.701,160.105
C08598=1015.155,171.609,373.838,167.092,54.713,160.106
C08599=1015.151,171.360,373.858,167.087,54.723,160.107
C08600=1015.146,171.080,373.882,167.083,54.736,160.109
C08601=1015.141,170.800,373.904,167.079,54.748,160.110
C08602=1015.137,170.520,373.927,167.074,54.761,160.112
C08603=1015.131,170.240,373.950,167.070,54.773,160.114
C08604=1015.127,169.991,373.971,167.066,54.785,160.115
C08605=1015.122,169.742,373.991,167.062,54.795,160.116
C08606=1015.118,169.493,374.011,167.058,54.807,160.118
C08607=1015.115,169.244,374.032,167.054,54.818,160.119
C08608=1015.110,168.994,374.052,167.050,54.829,160.120
C08609=1015.106,168.745,374.073,167.047,54.840,160.122
C08610=1015.101,168.496,374.092,167.044,54.851,160.123
C08611=1015.097,168.247,374.113,167.039,54.862,160.125
C08612=1015.092,167.998,374.134,167.036,54.873,160.126
C08613=1015.089,167.749,374.154,167.031,54.884,160.127
C08614=1015.084,167.500,374.175,167.028,54.895,160.129
C08615=1015.080,167.251,374.194,167.025,54.906,160.130
C08616=1015.076,167.002,374.215,167.021,54.917,160.132
C08617=1015.071,166.752,374.235,167.017,54.929,160.133
C08618=1015.067,166.503,374.256,167.013,54.939,160.134
C08619=1015.063,166.254,374.276,167.009,54.951,160.136
C08620=1015.058,166.005,374.296,167.005,54.961,160.137
C08621=1015.054,165.756,374.316,167.002,54.972,160.139
C08622=1015.050,165.507,374.336,166.998,54.984,160.140
C08623=1015.046,165.257,374.357,166.994,54.995,160.141
C08624=1015.041,165.008,374.377,166.990,55.006,160.143
C08625=1015.037,164.759,374.397,166.987,55.016,160.144
C08626=1015.034,164.510,374.417,166.983,55.028,160.146
C08627=1015.028,164.261,374.438,166.979,55.038,160.147
C08628=1015.025,164.012,374.458,166.975,55.050,160.148
C08629=1015.020,163.762,374.477,166.971,55.061,160.149
C08630=1015.017,163.514,374.498,166.968,55.072,160.151
C08631=1015.012,163.264,374.518,166.964,55.082,160.152
C08632=1015.008,163.015,374.539,166.961,55.094,160.154
C08633=1015.004,162.766,374.559,166.958,55.105,160.155
C08634=1015.000,162.517,374.578,166.954,55.116,160.157
C08635=1014.995,162.267,374.600,166.950,55.127,160.158
C08636=1014.991,162.018,374.619,166.946,55.138,160.159
C08637=1014.987,161.769,374.639,166.943,55.149,160.161
C08638=1014.983,161.520,374.660,166.939,55.160,160.162
C08639=1014.979,161.271,374.679,166.935,55.171,160.164
C08640=1014.975,161.021,374.700,166.932,55.182,160.165
C08641=1014.970,160.773,374.720,166.928,55.193,160.166
C08642=1014.966,160.523,374.740,166.924,55.204,160.168
C08643=1014.962,160.274,374.759,166.922,55.215,160.169
C08644=1014.958,160.026,374.780,166.917,55.226,160.170
C08645=1014.955,159.776,374.800,166.913,55.236,160.172
C08646=1014.950,159.527,374.820,166.911,55.247,160.173
C08647=1014.946,159.278,374.841,166.906,55.258,160.175
C08648=1014.941,159.029,374.860,166.903,55.270,160.176
C08649=1014.938,158.779,374.880,166.900,55.280,160.177
C08650=1014.934,158.530,374.901,166.896,55.292,160.179
C08651=1014.929,158.280,374.920,166.892,55.302,160.180
C08652=1014.925,158.031,374.940,166.889,55.313,160.182
C08653=1014.921,157.782,374.959,166.886,55.325,160.183
C08654=1014.916,157.533,374.979,166.882,55.336,160.184
C08655=1014.913,157.284,374.999,166.878,55.347,160.186
C08656=1014.908,157.035,375.018,166.874,55.359,160.187
C08657=1014.903,156.785,375.038,166.871,55.369,160.189
C08658=1014.899,156.536,375.058,166.868,55.381,160.190
C08659=1014.895,156.287,375.077,166.864,55.392,160.192
C08660=1014.890,156.038,375.097,166.860,55.403,160.193
C08661=1014.886,155.789,375.116,166.857,55.414,160.195
C08662=1014.882,155.540,375.136,166.854,55.426,160.196
C08663=1014.877,155.291,375.155,166.849,55.436,160.197
C08664=1014.872,155.010,375.177,166.845,55.449,160.199
C08665=1014.868,154.730,375.199,166.841,55.462,160.200
C08666=1014.862,154.450,375.221,166.838,55.474,160.202
C08667=1014.858,154.169,375.243,166.834,55.487,160.204
C08668=1014.853,153.920,375.262,166.830,55.498,160.205
C08669=1014.849,153.671,375.282,166.826,55.509,160.207
C08670=1014.845,153.422,375.300,166.824,55.520,160.208
C08671=1014.841,153.173,375.320,166.820,55.532,160.210
C08672=1014.837,152.923,375.340,166.816,55.542,160.211
C08673=1014.833,152.674,375.359,166.814,55.553,160.213
C08674=1014.828,152.425,375.379,166.810,55.565,160.214
C08675=1014.824,152.175,375.398,166.806,55.576,160.215
C08676=1014.819,151.926,375.418,166.803,55.587,160.217
C08677=1014.815,151.677,375.437,166.800,55.599,160.218
C08678=1014.810,151.428,375.456,166.796,55.609,160.220
C08679=1014.806,151.178,375.475,166.792,55.621,160.221
C08680=1014.802,150.929,375.494,166.790,55.632,160.223
C08681=1014.797,150.680,375.514,166.786,55.643,160.224
C08682=1014.793,150.431,375.533,166.782,55.654,160.225
C08683=1014.789,150.181,375.552,166.779,55.665,160.227
C08684=1014.785,149.932,375.571,166.776,55.677,160.228
C08685=1014.780,149.683,375.591,166.772,55.688,160.230
C08686=1014.776,149.434,375.610,166.769,55.699,160.231
C08687=1014.772,149.185,375.629,166.765,55.710,160.233
C08688=1014.767,148.936,375.648,166.762,55.722,160.234
C08689=1014.763,148.686,375.667,166.759,55.732,160.236
C08690=1014.759,148.437,375.687,166.755,55.744,160.237
C08691=1014.755,148.187,375.705,166.751,55.755,160.238
C08692=1014.751,147.938,375.725,166.749,55.766,160.240
C08693=1014.746,147.689,375.744,166.745,55.777,160.242
C08694=1014.742,147.440,375.763,166.741,55.788,160.243
C08695=1014.738,147.191,375.782,166.739,55.799,160.244
C08696=1014.734,146.942,375.800,166.735,55.810,160.246
C08697=1014.729,146.693,375.820,166.732,55.821,160.247
C08698=1014.725,146.443,375.839,166.729,55.833,160.249
C08699=1014.721,146.194,375.858,166.725,55.844,160.250
C08700=1014.717,145.945,375.878,166.722,55.855,160.252
C08701=1014.712,145.696,375.896,166.718,55.866,160.253
C08702=1014.708,145.447,375.915,166.715,55.878,160.254
C08703=1014.703,145.197,375.934,166.712,55.889,160.256
C08704=1014.699,144.947,375.953,166.708,55.900,160.257
C08705=1014.694,144.699,375.972,166.705,55.911,160.259
C08706=1014.690,144.449,375.990,166.703,55.922,160.261
C08707=1014.686,144.200,376.010,166.699,55.933,160.262
C08708=1014.681,143.951,376.028,166.696,55.945,160.263
C08709=1014.678,143.702,376.046,166.693,55.956,160.265
C08710=1014.673,143.453,376.066,166.689,55.967,160.266
C08711=1014.669,143.203,376.084,166.686,55.978,160.268
C08712=1014.665,142.954,376.103,166.682,55.989,160.269
C08713=1014.660,142.704,376.122,166.679,56.001,160.271
C08714=1014.655,142.455,376.140,166.676,56.012,160.272
C08715=1014.651,142.205,376.159,166.672,56.023,160.274
C08716=1014.647,141.956,376.179,166.670,56.034,160.275
C08717=1014.643,141.708,376.196,166.666,56.045,160.277
C08718=1014.639,141.458,376.215,166.663,56.057,160.278
C08719=1014.634,141.209,376.235,166.660,56.068,160.280
C08720=1014.630,140.960,376.253,166.656,56.079,160.281
C08721=1014.626,140.710,376.272,166.654,56.090,160.283
C08722=1014.621,140.461,376.290,166.650,56.101,160.284
C08723=1014.617,140.212,376.309,166.647,56.113,160.285
C08724=1014.613,139.963,376.328,166.644,56.123,160.287
C08725=1014.608,139.713,376.346,166.640,56.135,160.288
C08726=1014.604,139.464,376.365,166.638,56.146,160.290
C08727=1014.600,139.215,376.384,166.634,56.157,160.291
C08728=1014.595,138.935,376.405,166.631,56.169,160.293
C08729=1014.591,138.654,376.426,166.627,56.182,160.295
C08730=1014.585,138.374,376.447,166.624,56.195,160.297
C08731=1014.580,138.094,376.467,166.620,56.207,160.298
C08732=1014.576,137.845,376.487,166.617,56.218,160.299
C08733=1014.573,137.596,376.505,166.614,56.229,160.301
C08734=1014.568,137.346,376.523,166.610,56.241,160.302
C08735=1014.564,137.097,376.542,166.608,56.252,160.304
C08736=1014.559,136.847,376.560,166.604,56.263,160.305
C08737=1014.555,136.598,376.579,166.602,56.274,160.307
C08738=1014.551,136.349,376.597,166.598,56.285,160.308
C08739=1014.547,136.099,376.615,166.596,56.296,160.310
C08740=1014.542,135.850,376.633,166.592,56.307,160.311
C08741=1014.538,135.600,376.652,166.589,56.319,160.313
C08742=1014.534,135.352,376.670,166.586,56.330,160.314
C08743=1014.529,135.102,376.688,166.583,56.341,160.316
C08744=1014.525,134.853,376.707,166.580,56.353,160.317
C08745=1014.520,134.603,376.725,166.576,56.364,160.319
C08746=1014.517,134.354,376.744,166.574,56.375,160.320
C08747=1014.512,134.105,376.762,166.570,56.386,160.322
C08748=1014.507,133.856,376.780,166.567,56.397,160.323
C08749=1014.503,133.606,376.799,166.564,56.408,160.325
C08750=1014.499,133.357,376.816,166.561,56.419,160.326
C08751=1014.495,133.108,376.835,166.557,56.430,160.327
C08752=1014.490,132.858,376.853,166.555,56.442,160.329
C08753=1014.486,132.610,376.871,166.551,56.453,160.330
C08754=1014.482,132.360,376.890,166.549,56.464,160.332
C08755=1014.477,132.111,376.908,166.545,56.475,160.333
C08756=1014.472,131.861,376.926,166.543,56.486,160.335
C08757=1014.469,131.612,376.945,166.540,56.497,160.337
C08758=1014.464,131.363,376.963,166.537,56.509,160.338
C08759=1014.460,131.113,376.981,166.534,56.519,160.340
C08760=1014.456,130.865,376.999,166.531,56.531,160.341
C08761=1014.451,130.615,377.017,166.528,56.541,160.343
C08762=1014.447,130.365,377.035,166.525,56.553,160.344
C08763=1014.443,130.116,377.053,166.522,56.564,160.346
C08764=1014.439,129.867,377.072,166.518,56.576,160.347
C08765=1014.434,129.617,377.090,166.516,56.586,160.349
C08766=1014.430,129.369,377.108,166.513,56.597,160.350
C08767=1014.426,129.119,377.125,166.510,56.608,160.351
C08768=1014.421,128.869,377.144,166.507,56.620,160.353
C08769=1014.417,128.621,377.161,166.504,56.631,160.354
C08770=1014.413,128.370,377.179,166.500,56.643,160.356
C08771=1014.408,128.121,377.198,166.498,56.653,160.357
C08772=1014.404,127.872,377.215,166.494,56.665,160.359
C08773=1014.400,127.622,377.233,166.492,56.676,160.361
C08774=1014.395,127.373,377.251,166.488,56.687,160.362
C08775=1014.391,127.124,377.269,166.486,56.699,160.364
C08776=1014.386,126.874,377.286,166.482,56.710,160.365
C08777=1014.382,126.626,377.304,166.480,56.721,160.367
C08778=1014.378,126.376,377.321,166.476,56.732,160.368
C08779=1014.373,126.127,377.340,166.474,56.743,160.370
C08780=1014.369,125.878,377.357,166.471,56.754,160.371
C08781=1014.364,125.628,377.375,166.468,56.766,160.373
C08782=1014.360,125.379,377.393,166.465,56.776,160.374
C08783=1014.355,125.129,377.410,166.462,56.788,160.376
C08784=1014.351,124.880,377.428,166.459,56.799,160.377
C08785=1014.347,124.631,377.445,166.456,56.811,160.379
C08786=1014.342,124.381,377.464,166.454,56.821,160.380
C08787=1014.338,124.133,377.481,166.450,56.833,160.382
C08788=1014.333,123.883,377.499,166.448,56.844,160.383
C08789=1014.329,123.633,377.517,166.445,56.855,160.385
C08790=1014.325,123.384,377.534,166.442,56.866,160.386
C08791=1014.320,123.135,377.552,166.440,56.877,160.388
C08792=1014.316,122.855,377.572,166.435,56.890,160.389
C08793=1014.310,122.574,377.591,166.433,56.902,160.391
C08794=1014.305,122.294,377.611,166.429,56.915,160.393
C08795=1014.301,122.014,377.631,166.426,56.927,160.395
C08796=1014.296,121.765,377.649,166.424,56.938,160.396
C08797=1014.292,121.515,377.666,166.420,56.949,160.398
C08798=1014.288,121.265,377.684,166.417,56.960,160.399
C08799=1014.284,121.017,377.702,166.415,56.972,160.401
C08800=1014.279,120.767,377.719,166.412,56.983,160.402
C08801=1014.275,120.518,377.737,166.409,56.993,160.403
C08802=1014.271,120.268,377.754,166.407,57.005,160.405
C08803=1014.267,120.019,377.772,166.403,57.016,160.407
C08804=1014.262,119.769,377.790,166.400,57.026,160.408
C08805=1014.258,119.521,377.807,166.398,57.038,160.410
C08806=1014.253,119.271,377.825,166.395,57.049,160.411
C08807=1014.249,119.022,377.843,166.392,57.060,160.413
C08808=1014.245,118.772,377.860,166.390,57.071,160.414
C08809=1014.241,118.523,377.877,166.387,57.082,160.416
C08810=1014.236,118.274,377.895,166.383,57.093,160.417
C08811=1014.232,118.024,377.912,166.381,57.103,160.418
C08812=1014.227,117.775,377.931,166.379,57.115,160.420
C08813=1014.224,117.526,377.948,166.376,57.126,160.422
C08814=1014.219,117.276,377.965,166.372,57.137,160.423
C08815=1014.215,117.027,377.983,166.370,57.147,160.424
C08816=1014.210,116.777,378.000,166.368,57.159,160.426
C08817=1014.206,116.528,378.018,166.365,57.169,160.428
C08818=1014.202,116.279,378.035,166.361,57.181,160.429
C08819=1014.198,116.029,378.053,166.359,57.191,160.431
C08820=1014.194,115.781,378.070,166.356,57.202,160.432
C08821=1014.189,115.531,378.088,166.354,57.213,160.434
C08822=1014.185,115.281,378.105,166.352,57.224,160.435
C08823=1014.181,115.032,378.123,166.348,57.235,160.437
C08824=1014.177,114.783,378.140,166.345,57.246,160.438
C08825=1014.173,114.533,378.157,166.343,57.257,160.439
C08826=1014.168,114.284,378.175,166.340,57.267,160.441
C08827=1014.164,114.035,378.193,166.337,57.278,160.442
C08828=1014.160,113.785,378.210,166.334,57.290,160.444
C08829=1014.156,113.536,378.228,166.332,57.301,160.446
C08830=1014.152,113.287,378.245,166.329,57.311,160.447
C08831=1014.147,113.037,378.262,166.327,57.322,160.449
C08832=1014.143,112.788,378.279,166.324,57.333,160.450
C08833=1014.139,112.539,378.297,166.321,57.344,160.451
C08834=1014.135,112.289,378.315,166.319,57.354,160.453
C08835=1014.131,112.040,378.332,166.316,57.365,160.454
C08836=1014.126,111.790,378.350,166.313,57.376,160.456
C08837=1014.122,111.541,378.367,166.310,57.387,160.457
C08838=1014.118,111.292,378.383,166.308,57.398,160.459
C08839=1014.113,111.042,378.401,166.306,57.409,160.461
C08840=1014.109,110.793,378.418,166.303,57.420,160.462
C08841=1014.105,110.544,378.435,166.299,57.431,160.463
C08842=1014.100,110.294,378.452,166.297,57.442,160.465
C08843=1014.096,110.045,378.469,166.294,57.452,160.466
C08844=1014.092,109.795,378.486,166.292,57.463,160.468
C08845=1014.087,109.546,378.503,166.290,57.475,160.470
C08846=1014.083,109.297,378.520,166.287,57.485,160.471
C08847=1014.079,109.047,378.537,166.284,57.497,160.472
C08848=1014.074,108.798,378.554,166.281,57.507,160.474
C08849=1014.070,108.548,378.571,166.279,57.518,160.475
C08850=1014.066,108.299,378.587,166.276,57.529,160.477
C08851=1014.061,108.049,378.605,166.274,57.540,160.479
C08852=1014.057,107.800,378.621,166.271,57.552,160.480
C08853=1014.053,107.551,378.638,166.268,57.562,160.482
C08854=1014.048,107.302,378.655,166.265,57.573,160.483
C08855=1014.044,107.052,378.672,166.263,57.584,160.485
C08856=1014.039,106.772,378.691,166.261,57.596,160.486
C08857=1014.034,106.491,378.710,166.257,57.609,160.488
C08858=1014.029,106.211,378.729,166.254,57.621,160.489
C08859=1014.024,105.932,378.748,166.251,57.633,160.491
C08860=1014.020,105.683,378.765,166.249,57.644,160.493
C08861=1014.015,105.432,378.781,166.246,57.655,160.494
C08862=1014.011,105.183,378.798,166.244,57.666,160.496
C08863=1014.007,104.934,378.815,166.241,57.677,160.497
C08864=1014.003,104.685,378.832,166.239,57.687,160.499
C08865=1013.998,104.435,378.849,166.235,57.699,160.500
C08866=1013.994,104.186,378.866,166.233,57.709,160.502
C08867=1013.989,103.937,378.882,166.230,57.720,160.503
C08868=1013.985,103.687,378.898,166.228,57.731,160.505
C08869=1013.980,103.437,378.915,166.225,57.742,160.506
C08870=1013.976,103.188,378.932,166.223,57.752,160.508
C08871=1013.972,102.939,378.949,166.220,57.763,160.509
C08872=1013.968,102.690,378.966,166.218,57.774,160.511
C08873=1013.963,102.440,378.982,166.216,57.785,160.512
C08874=1013.959,102.190,378.999,166.213,57.796,160.514
C08875=1013.954,101.941,379.016,166.211,57.806,160.515
C08876=1013.951,101.692,379.033,166.208,57.817,160.517
C08877=1013.945,101.442,379.050,166.206,57.828,160.518
C08878=1013.942,101.193,379.066,166.203,57.838,160.520
C08879=1013.937,100.944,379.082,166.200,57.849,160.521
C08880=1013.933,100.694,379.100,166.198,57.860,160.523
C08881=1013.929,100.445,379.116,166.195,57.871,160.524
C08882=1013.925,100.195,379.133,166.193,57.881,160.526
C08883=1013.921,99.945,379.150,166.190,57.892,160.527
C08884=1013.916,99.697,379.166,166.188,57.903,160.529
C08885=1013.912,99.447,379.183,166.185,57.913,160.530
C08886=1013.908,99.198,379.199,166.183,57.924,160.532
C08887=1013.904,98.948,379.216,166.180,57.935,160.533
C08888=1013.899,98.699,379.233,166.178,57.946,160.535
C08889=1013.895,98.449,379.249,166.175,57.956,160.536
C08890=1013.890,98.200,379.265,166.173,57.967,160.538
C08891=1013.886,97.950,379.282,166.171,57.978,160.539
C08892=1013.882,97.701,379.298,166.168,57.989,160.541
C08893=1013.877,97.452,379.315,166.166,58.000,160.542
C08894=1013.872,97.202,379.331,166.163,58.010,160.544
C08895=1013.868,96.953,379.347,166.160,58.021,160.545
C08896=1013.864,96.703,379.364,166.158,58.031,160.547
C08897=1013.859,96.454,379.380,166.156,58.042,160.548
C08898=1013.855,96.205,379.396,166.153,58.053,160.550
C08899=1013.850,95.956,379.412,166.151,58.064,160.551
C08900=1013.846,95.705,379.429,166.148,58.075,160.553
C08901=1013.842,95.456,379.446,166.146,58.086,160.554
C08902=1013.837,95.207,379.461,166.143,58.096,160.556
C08903=1013.833,94.958,379.478,166.141,58.107,160.557
C08904=1013.828,94.708,379.494,166.138,58.117,160.559
C08905=1013.825,94.459,379.511,166.136,58.128,160.560
C08906=1013.820,94.209,379.526,166.134,58.139,160.562
C08907=1013.816,93.960,379.542,166.131,58.149,160.563
C08908=1013.811,93.710,379.559,166.128,58.160,160.564
C08909=1013.806,93.460,379.575,166.126,58.171,160.566
C08910=1013.803,93.211,379.592,166.123,58.181,160.567
C08911=1013.798,92.962,379.608,166.122,58.191,160.569
C08912=1013.794,92.713,379.624,166.119,58.202,160.571
C08913=1013.789,92.463,379.640,166.117,58.213,160.572
C08914=1013.785,92.214,379.656,166.114,58.223,160.573
C08915=1013.781,91.964,379.673,166.112,58.234,160.575
C08916=1013.777,91.715,379.689,166.110,58.245,160.576
C08917=1013.772,91.466,379.705,166.107,58.255,160.578
C08918=1013.768,91.216,379.721,166.105,58.266,160.579
C08919=1013.763,90.967,379.737,166.103,58.276,160.581
C08920=1013.759,90.687,379.756,166.100,58.288,160.582
C08921=1013.754,90.406,379.774,166.097,58.300,160.584
C08922=1013.749,90.127,379.792,166.094,58.312,160.586
C08923=1013.745,89.847,379.810,166.092,58.324,160.588
C08924=1013.740,89.598,379.826,166.090,58.334,160.589
C08925=1013.736,89.349,379.842,166.087,58.345,160.590
C08926=1013.731,89.099,379.858,166.084,58.355,160.592
C08927=1013.728,88.850,379.875,166.083,58.365,160.593
C08928=1013.723,88.600,379.891,166.080,58.375,160.595
C08929=1013.719,88.351,379.907,166.078,58.386,160.596
C08930=1013.714,88.100,379.923,166.076,58.397,160.598
C08931=1013.709,87.852,379.939,166.073,58.407,160.599
C08932=1013.704,87.602,379.954,166.070,58.418,160.601
C08933=1013.700,87.353,379.970,166.069,58.429,160.602
C08934=1013.696,87.103,379.986,166.066,58.439,160.604
C08935=1013.691,86.853,380.002,166.064,58.450,160.605
C08936=1013.687,86.604,380.018,166.061,58.460,160.606
C08937=1013.683,86.354,380.033,166.059,58.471,160.608
C08938=1013.678,86.105,380.050,166.057,58.482,160.610
C08939=1013.674,85.856,380.066,166.055,58.491,160.611
C08940=1013.669,85.606,380.081,166.053,58.502,160.613
C08941=1013.665,85.357,380.096,166.050,58.512,160.614
C08942=1013.660,85.107,380.112,166.047,58.523,160.615
C08943=1013.656,84.858,380.128,166.045,58.534,160.617
C08944=1013.652,84.608,380.144,166.043,58.544,160.618
C08945=1013.647,84.359,380.160,166.041,58.554,160.620
C08946=1013.644,84.110,380.175,166.038,58.565,160.621
C08947=1013.639,83.861,380.191,166.035,58.575,160.623
C08948=1013.634,83.612,380.207,166.034,58.586,160.624
C08949=1013.630,83.362,380.222,166.031,58.596,160.626
C08950=1013.625,83.112,380.238,166.029,58.606,160.627
C08951=1013.621,82.863,380.254,166.027,58.617,160.629
C08952=1013.617,82.613,380.270,166.025,58.627,160.630
C08953=1013.612,82.364,380.285,166.022,58.638,160.632
C08954=1013.608,82.114,380.301,166.021,58.647,160.633
C08955=1013.604,81.864,380.317,166.018,58.658,160.634
C08956=1013.599,81.615,380.332,166.016,58.669,160.636
C08957=1013.595,81.366,380.348,166.014,58.678,160.637
C08958=1013.590,81.116,380.364,166.011,58.689,160.639
C08959=1013.586,80.866,380.379,166.009,58.699,160.640
C08960=1013.582,80.617,380.395,166.007,58.709,160.642
C08961=1013.577,80.367,380.411,166.004,58.719,160.643
C08962=1013.574,80.118,380.426,166.002,58.730,160.644
C08963=1013.569,79.869,380.442,166.000,58.740,160.646
C08964=1013.564,79.620,380.457,165.997,58.750,160.647
C08965=1013.560,79.370,380.473,165.996,58.760,160.649
C08966=1013.556,79.120,380.489,165.994,58.771,160.650
C08967=1013.551,78.871,380.505,165.992,58.781,160.652
C08968=1013.547,78.621,380.520,165.989,58.791,160.653
C08969=1013.543,78.372,380.536,165.986,58.801,160.654
C08970=1013.538,78.122,380.552,165.984,58.811,160.656
C08971=1013.534,77.873,380.568,165.982,58.822,160.657
C08972=1013.530,77.624,380.583,165.981,58.832,160.659
C08973=1013.525,77.374,380.598,165.978,58.842,160.660
C08974=1013.521,77.125,380.614,165.976,58.852,160.662
C08975=1013.517,76.875,380.630,165.973,58.862,160.663
C08976=1013.512,76.626,380.646,165.972,58.872,160.664
C08977=1013.508,76.375,380.661,165.969,58.882,160.666
C08978=1013.503,76.126,380.676,165.968,58.893,160.668
C08979=1013.499,75.877,380.692,165.965,58.903,160.669
C08980=1013.495,75.628,380.707,165.963,58.913,160.670
C08981=1013.490,75.378,380.722,165.960,58.923,160.672
C08982=1013.486,75.128,380.737,165.958,58.933,160.673
C08983=1013.482,74.879,380.753,165.956,58.943,160.674
C08984=1013.476,74.600,380.770,165.953,58.955,160.676
C08985=1013.471,74.320,380.787,165.951,58.966,160.678
C08986=1013.467,74.040,380.804,165.949,58.977,160.679
C08987=1013.462,73.761,380.822,165.946,58.988,160.681
C08988=1013.457,73.511,380.836,165.944,58.998,160.682
C08989=1013.453,73.261,380.852,165.942,59.008,160.683
C08990=1013.448,73.013,380.867,165.940,59.018,160.685
C08991=1013.444,72.763,380.882,165.938,59.029,160.687
C08992=1013.440,72.513,380.898,165.936,59.039,160.688
C08993=1013.435,72.264,380.913,165.933,59.049,160.689
C08994=1013.431,72.014,380.928,165.932,59.059,160.691
C08995=1013.427,71.765,380.943,165.929,59.069,160.692
C08996=1013.422,71.515,380.959,165.927,59.079,160.694
C08997=1013.417,71.266,380.974,165.925,59.089,160.695
C08998=1013.413,71.016,380.989,165.922,59.098,160.696
C08999=1013.409,70.766,381.005,165.921,59.108,160.698
C09000=1013.404,70.518,381.019,165.918,59.119,160.699
C09001=1013.400,70.268,381.034,165.916,59.128,160.700
C09002=1013.395,70.018,381.050,165.914,59.139,160.702
C09003=1013.391,69.768,381.065,165.912,59.148,160.703
C09004=1013.387,69.520,381.079,165.910,59.158,160.705
C09005=1013.383,69.270,381.095,165.908,59.169,160.706
C09006=1013.378,69.020,381.110,165.906,59.178,160.708
C09007=1013.374,68.771,381.125,165.904,59.188,160.709
C09008=1013.370,68.520,381.140,165.901,59.198,160.710
C09009=1013.365,68.272,381.155,165.899,59.208,160.712
C09010=1013.361,68.022,381.171,165.898,59.217,160.713
C09011=1013.356,67.772,381.186,165.895,59.228,160.714
C09012=1013.352,67.523,381.201,165.893,59.237,160.716
C09013=1013.348,67.274,381.215,165.892,59.247,160.717
C09014=1013.343,67.024,381.231,165.888,59.257,160.718
C09015=1013.339,66.774,381.246,165.887,59.267,160.720
C09016=1013.334,66.525,381.261,165.885,59.277,160.721
C09017=1013.330,66.276,381.275,165.883,59.287,160.723
C09018=1013.325,66.026,381.291,165.881,59.297,160.724
C09019=1013.320,65.776,381.305,165.879,59.306,160.725
C09020=1013.317,65.527,381.321,165.876,59.316,160.727
C09021=1013.312,65.277,381.335,165.874,59.326,160.728
C09022=1013.307,65.027,381.349,165.873,59.336,160.730
C09023=1013.303,64.778,381.365,165.871,59.345,160.731
C09024=1013.299,64.529,381.379,165.868,59.355,160.732
C09025=1013.294,64.279,381.394,165.866,59.365,160.734
C09026=1013.290,64.029,381.410,165.864,59.374,160.735
C09027=1013.286,63.780,381.424,165.863,59.384,160.737
C09028=1013.281,63.531,381.439,165.860,59.394,160.738
C09029=1013.277,63.281,381.454,165.858,59.403,160.739
C09030=1013.272,63.032,381.469,165.856,59.413,160.741
C09031=1013.267,62.782,381.483,165.855,59.423,160.742
C09032=1013.263,62.532,381.498,165.851,59.433,160.743
C09033=1013.259,62.283,381.513,165.850,59.442,160.745
C09034=1013.254,62.034,381.527,165.848,59.452,160.746
C09035=1013.250,61.784,381.542,165.846,59.461,160.747
C09036=1013.245,61.534,381.556,165.843,59.472,160.749
C09037=1013.241,61.285,381.570,165.842,59.482,160.750
C09038=1013.236,61.035,381.586,165.840,59.491,160.751
C09039=1013.231,60.786,381.600,165.838,59.501,160.753
C09040=1013.227,60.536,381.614,165.835,59.511,160.754
C09041=1013.222,60.286,381.629,165.833,59.520,160.756
C09042=1013.218,60.037,381.643,165.832,59.530,160.757
C09043=1013.213,59.787,381.657,165.829,59.539,160.758
C09044=1013.208,59.537,381.672,165.827,59.549,160.760
C09045=1013.204,59.289,381.686,165.825,59.559,160.761
C09046=1013.199,59.039,381.701,165.823,59.568,160.762
C09047=1013.195,58.790,381.715,165.822,59.578,160.764
C09048=1013.190,58.510,381.731,165.819,59.589,160.765
C09049=1013.185,58.230,381.747,165.817,59.600,160.767
C09050=1013.180,57.951,381.764,165.814,59.610,160.768
C09051=1013.175,57.671,381.780,165.813,59.621,160.770
C09052=1013.170,57.421,381.795,165.810,59.630,160.771
C09053=1013.166,57.172,381.809,165.809,59.640,160.773
C09054=1013.161,56.922,381.823,165.807,59.649,160.774
C09055=1013.157,56.673,381.837,165.803,59.659,160.775
C09056=1013.152,56.423,381.852,165.802,59.669,160.776
C09057=1013.148,56.173,381.866,165.800,59.678,160.778
C09058=1013.144,55.924,381.880,165.798,59.688,160.779
C09059=1013.139,55.674,381.895,165.796,59.697,160.780
C09060=1013.134,55.426,381.910,165.794,59.706,160.782
C09061=1013.130,55.176,381.924,165.792,59.715,160.783
C09062=1013.126,54.927,381.938,165.790,59.725,160.784
C09063=1013.121,54.677,381.953,165.788,59.734,160.786
C09064=1013.117,54.428,381.967,165.786,59.743,160.787
C09065=1013.112,54.178,381.981,165.785,59.753,160.788
C09066=1013.107,53.928,381.996,165.782,59.762,160.790
C09067=1013.103,53.679,382.010,165.780,59.772,160.791
C09068=1013.098,53.429,382.024,165.778,59.781,160.792
C09069=1013.094,53.180,382.038,165.776,59.790,160.793
C09070=1013.089,52.930,382.053,165.775,59.800,160.795
C09071=1013.085,52.681,382.067,165.773,59.809,160.796
C09072=1013.081,52.431,382.081,165.771,59.818,160.797
C09073=1013.076,52.181,382.095,165.769,59.827,160.799
C09074=1013.072,51.932,382.110,165.767,59.836,160.800
C09075=1013.068,51.682,382.124,165.765,59.845,160.801
C09076=1013.063,51.432,382.138,165.763,59.854,160.802
C09077=1013.059,51.183,382.152,165.761,59.864,160.804
C09078=1013.054,50.933,382.167,165.759,59.873,160.805
C09079=1013.050,50.684,382.181,165.758,59.881,160.806
C09080=1013.045,50.434,382.195,165.755,59.891,160.807
C09081=1013.041,50.185,382.209,165.753,59.900,160.809
C09082=1013.036,49.935,382.224,165.751,59.909,160.810
C09083=1013.032,49.686,382.238,165.749,59.918,160.811
C09084=1013.027,49.436,382.253,165.748,59.927,160.813
C09085=1013.023,49.187,382.267,165.746,59.936,160.814
C09086=1013.018,48.937,382.281,165.744,59.945,160.815
C09087=1013.014,48.688,382.295,165.742,59.954,160.816
C09088=1013.010,48.438,382.310,165.741,59.963,160.818
C09089=1013.005,48.189,382.324,165.739,59.972,160.819
C09090=1013.001,47.938,382.337,165.736,59.981,160.820
C09091=1012.997,47.689,382.352,165.734,59.990,160.821
C09092=1012.992,47.439,382.366,165.733,59.999,160.823
C09093=1012.988,47.190,382.380,165.731,60.008,160.824
C09094=1012.983,46.940,382.395,165.729,60.017,160.825
C09095=1012.979,46.691,382.409,165.727,60.025,160.826
C09096=1012.975,46.442,382.423,165.725,60.034,160.827
C09097=1012.970,46.192,382.437,165.723,60.043,160.829
C09098=1012.966,45.943,382.451,165.721,60.051,160.830
C09099=1012.961,45.693,382.466,165.719,60.061,160.831
C09100=1012.957,45.444,382.480,165.718,60.069,160.832
C09101=1012.953,45.193,382.494,165.715,60.078,160.833
C09102=1012.949,44.944,382.508,165.713,60.087,160.835
C09103=1012.944,44.695,382.522,165.712,60.096,160.836
C09104=1012.940,44.445,382.536,165.709,60.104,160.837
C09105=1012.936,44.196,382.550,165.708,60.113,160.838
C09106=1012.931,43.946,382.565,165.706,60.121,160.839
C09107=1012.927,43.697,382.579,165.705,60.130,160.841
C09108=1012.923,43.448,382.593,165.703,60.139,160.842
C09109=1012.918,43.197,382.607,165.701,60.147,160.843
C09110=1012.914,42.948,382.621,165.699,60.157,160.844
C09111=1012.909,42.698,382.635,165.697,60.165,160.845
C09112=1012.903,42.319,382.657,165.694,60.177,160.847
